   1:  PR[GP1:91,1] = PR[GP1:90,1] + 48.175;
   1:  PR[GP1:91,2] = PR[GP1:90,2] + 18.982;
   1:L PR[91] 10mm/sec CNT100;
   1:  PR[GP1:91,1] = PR[GP1:90,1] + 43.044;
   1:  PR[GP1:91,2] = PR[GP1:90,2] + 27.550;
   1:L PR[91] 10mm/sec CNT100;
   1:  PR[GP1:91,1] = PR[GP1:90,1] + 39.834;
   1:  PR[GP1:91,2] = PR[GP1:90,2] + 31.417;
   1:L PR[91] 10mm/sec CNT100;
   1:  PR[GP1:91,1] = PR[GP1:90,1] + 32.306;
   1:  PR[GP1:91,2] = PR[GP1:90,2] + 37.456;
   1:L PR[91] 10mm/sec CNT100;
   1:  PR[GP1:91,1] = PR[GP1:90,1] + 28.401;
   1:  PR[GP1:91,2] = PR[GP1:90,2] + 40.222;
   1:L PR[91] 10mm/sec CNT100;
   1:  PR[GP1:91,1] = PR[GP1:90,1] + 23.934;
   1:  PR[GP1:91,2] = PR[GP1:90,2] + 41.952;
   1:L PR[91] 10mm/sec CNT100;
   1:  PR[GP1:91,1] = PR[GP1:90,1] + 14.950;
   1:  PR[GP1:91,2] = PR[GP1:90,2] + 44.976;
   1:L PR[91] 10mm/sec CNT100;
   1:  PR[GP1:91,1] = PR[GP1:90,1] + 9.867;
   1:  PR[GP1:91,2] = PR[GP1:90,2] + 45.606;
   1:L PR[91] 10mm/sec CNT100;
   1:  PR[GP1:91,1] = PR[GP1:90,1] + 0.933;
   1:  PR[GP1:91,2] = PR[GP1:90,2] + 45.414;
   1:L PR[91] 10mm/sec CNT100;
   1:  PR[GP1:91,1] = PR[GP1:90,1] + -0.069;
   1:  PR[GP1:91,2] = PR[GP1:90,2] + 45.753;
   1:  PR[GP1:91,3] = PR[GP1:90,3] + 114.380;
   1:L PR[91] 10mm/sec CNT100;
   1:  PR[GP1:91,1] = PR[GP1:90,1] + -8.239;
   1:  PR[GP1:91,2] = PR[GP1:90,2] + 45.929;
   1:L PR[91] 10mm/sec CNT100;
   1:  PR[GP1:91,1] = PR[GP1:90,1] + -13.918;
   1:  PR[GP1:91,2] = PR[GP1:90,2] + 45.225;
   1:L PR[91] 10mm/sec CNT100;
   1:  PR[GP1:91,1] = PR[GP1:90,1] + -22.131;
   1:  PR[GP1:91,2] = PR[GP1:90,2] + 42.461;
   1:L PR[91] 10mm/sec CNT100;
   1:  PR[GP1:91,1] = PR[GP1:90,1] + -27.169;
   1:  PR[GP1:91,2] = PR[GP1:90,2] + 40.508;
   1:L PR[91] 10mm/sec CNT100;
   1:  PR[GP1:91,1] = PR[GP1:90,1] + -34.286;
   1:  PR[GP1:91,2] = PR[GP1:90,2] + 34.822;
   1:L PR[91] 10mm/sec CNT100;
   1:  PR[GP1:91,1] = PR[GP1:90,1] + -38.499;
   1:  PR[GP1:91,2] = PR[GP1:90,2] + 31.839;
   1:L PR[91] 10mm/sec CNT100;
   1:  PR[GP1:91,1] = PR[GP1:90,1] + -42.170;
   1:  PR[GP1:91,2] = PR[GP1:90,2] + 27.417;
   1:L PR[91] 10mm/sec CNT100;
   1:  PR[GP1:91,1] = PR[GP1:90,1] + -46.861;
   1:  PR[GP1:91,2] = PR[GP1:90,2] + 19.580;
   1:L PR[91] 10mm/sec CNT100;
   1:  PR[GP1:91,1] = PR[GP1:90,1] + -49.099;
   1:  PR[GP1:91,2] = PR[GP1:90,2] + 14.512;
   1:L PR[91] 10mm/sec CNT100;
   1:  PR[GP1:91,1] = PR[GP1:90,1] + -50.765;
   1:  PR[GP1:91,2] = PR[GP1:90,2] + 5.371;
   1:L PR[91] 10mm/sec CNT100;
   1:  PR[GP1:91,1] = PR[GP1:90,1] + -51.513;
   1:  PR[GP1:91,2] = PR[GP1:90,2] + 0.008;
   1:L PR[91] 10mm/sec CNT100;
   1:  PR[GP1:91,1] = PR[GP1:90,1] + -49.864;
   1:  PR[GP1:91,2] = PR[GP1:90,2] + -9.008;
   1:L PR[91] 10mm/sec CNT100;
   1:  PR[GP1:91,1] = PR[GP1:90,1] + -49.094;
   1:  PR[GP1:91,2] = PR[GP1:90,2] + -14.532;
   1:L PR[91] 10mm/sec CNT100;
   1:  PR[GP1:91,1] = PR[GP1:90,1] + -46.862;
   1:  PR[GP1:91,2] = PR[GP1:90,2] + -19.588;
   1:L PR[91] 10mm/sec CNT100;
   1:  PR[GP1:91,1] = PR[GP1:90,1] + -42.171;
   1:  PR[GP1:91,2] = PR[GP1:90,2] + -27.425;
   1:L PR[91] 10mm/sec CNT100;
   1:  PR[GP1:91,1] = PR[GP1:90,1] + -38.488;
   1:  PR[GP1:91,2] = PR[GP1:90,2] + -31.861;
   1:L PR[91] 10mm/sec CNT100;
   1:  PR[GP1:91,1] = PR[GP1:90,1] + -31.608;
   1:  PR[GP1:91,2] = PR[GP1:90,2] + -37.380;
   1:L PR[91] 10mm/sec CNT100;
   1:  PR[GP1:91,1] = PR[GP1:90,1] + -27.187;
   1:  PR[GP1:91,2] = PR[GP1:90,2] + -40.510;
   1:L PR[91] 10mm/sec CNT100;
   1:  PR[GP1:91,1] = PR[GP1:90,1] + -22.133;
   1:  PR[GP1:91,2] = PR[GP1:90,2] + -42.469;
   1:L PR[91] 10mm/sec CNT100;
   1:  PR[GP1:91,1] = PR[GP1:90,1] + -13.920;
   1:  PR[GP1:91,2] = PR[GP1:90,2] + -45.233;
   1:L PR[91] 10mm/sec CNT100;
   1:  PR[GP1:91,1] = PR[GP1:90,1] + -8.241;
   1:  PR[GP1:91,2] = PR[GP1:90,2] + -45.937;
   1:L PR[91] 10mm/sec CNT100;
   1:  PR[GP1:91,1] = PR[GP1:90,1] + -0.070;
   1:  PR[GP1:91,2] = PR[GP1:90,2] + -45.762;
   1:L PR[91] 10mm/sec CNT100;
   1:  PR[GP1:91,1] = PR[GP1:90,1] + 0.889;
   1:L PR[91] 10mm/sec CNT100;
   1:  PR[GP1:91,1] = PR[GP1:90,1] + 9.061;
   1:  PR[GP1:91,2] = PR[GP1:90,2] + -45.937;
   1:L PR[91] 10mm/sec CNT100;
   1:  PR[GP1:91,1] = PR[GP1:90,1] + 14.741;
   1:  PR[GP1:91,2] = PR[GP1:90,2] + -45.234;
   1:L PR[91] 10mm/sec CNT100;
   1:  PR[GP1:91,1] = PR[GP1:90,1] + 22.954;
   1:  PR[GP1:91,2] = PR[GP1:90,2] + -42.469;
   1:L PR[91] 10mm/sec CNT100;
   1:  PR[GP1:91,1] = PR[GP1:90,1] + 27.992;
   1:  PR[GP1:91,2] = PR[GP1:90,2] + -40.516;
   1:L PR[91] 10mm/sec CNT100;
   1:  PR[GP1:91,1] = PR[GP1:90,1] + 35.108;
   1:  PR[GP1:91,2] = PR[GP1:90,2] + -34.829;
   1:L PR[91] 10mm/sec CNT100;
   1:  PR[GP1:91,1] = PR[GP1:90,1] + 39.322;
   1:  PR[GP1:91,2] = PR[GP1:90,2] + -31.845;
   1:L PR[91] 10mm/sec CNT100;
   1:  PR[GP1:91,1] = PR[GP1:90,1] + 42.992;
   1:  PR[GP1:91,2] = PR[GP1:90,2] + -27.423;
   1:L PR[91] 10mm/sec CNT100;
   1:  PR[GP1:91,1] = PR[GP1:90,1] + 47.683;
   1:  PR[GP1:91,2] = PR[GP1:90,2] + -19.591;
   1:L PR[91] 10mm/sec CNT100;
   1:  PR[GP1:91,1] = PR[GP1:90,1] + 49.920;
   1:  PR[GP1:91,2] = PR[GP1:90,2] + -14.523;
   1:L PR[91] 10mm/sec CNT100;
   1:  PR[GP1:91,1] = PR[GP1:90,1] + 51.586;
   1:  PR[GP1:91,2] = PR[GP1:90,2] + -5.380;
   1:L PR[91] 10mm/sec CNT100;
   1:  PR[GP1:91,1] = PR[GP1:90,1] + 52.334;
   1:  PR[GP1:91,2] = PR[GP1:90,2] + -0.017;
   1:L PR[91] 10mm/sec CNT100;
   1:  PR[GP1:91,1] = PR[GP1:90,1] + 50.685;
   1:  PR[GP1:91,2] = PR[GP1:90,2] + 9.003;
   1:L PR[91] 10mm/sec CNT100;
   1:  PR[GP1:91,1] = PR[GP1:90,1] + 49.914;
   1:  PR[GP1:91,2] = PR[GP1:90,2] + 14.527;
   1:L PR[91] 10mm/sec CNT100;
   1:  PR[GP1:91,1] = PR[GP1:90,1] + 47.682;
   1:  PR[GP1:91,2] = PR[GP1:90,2] + 19.583;
   1:L PR[91] 10mm/sec CNT100;
   1:  PR[GP1:91,1] = PR[GP1:90,1] + 42.991;
   1:  PR[GP1:91,2] = PR[GP1:90,2] + 27.415;
   1:L PR[91] 10mm/sec CNT100;
   1:  PR[GP1:91,1] = PR[GP1:90,1] + 39.310;
   1:  PR[GP1:91,2] = PR[GP1:90,2] + 31.851;
   1:L PR[91] 10mm/sec CNT100;
   1:  PR[GP1:91,1] = PR[GP1:90,1] + 32.429;
   1:  PR[GP1:91,2] = PR[GP1:90,2] + 37.371;
   1:L PR[91] 10mm/sec CNT100;
   1:  PR[GP1:91,1] = PR[GP1:90,1] + 28.007;
   1:  PR[GP1:91,2] = PR[GP1:90,2] + 40.502;
   1:L PR[91] 10mm/sec CNT100;
   1:  PR[GP1:91,1] = PR[GP1:90,1] + 22.952;
   1:  PR[GP1:91,2] = PR[GP1:90,2] + 42.461;
   1:L PR[91] 10mm/sec CNT100;
   1:  PR[GP1:91,1] = PR[GP1:90,1] + 14.739;
   1:  PR[GP1:91,2] = PR[GP1:90,2] + 45.225;
   1:L PR[91] 10mm/sec CNT100;
   1:  PR[GP1:91,1] = PR[GP1:90,1] + 9.059;
   1:  PR[GP1:91,2] = PR[GP1:90,2] + 45.928;
   1:L PR[91] 10mm/sec CNT100;
   1:  PR[GP1:91,1] = PR[GP1:90,1] + 0.889;
   1:  PR[GP1:91,2] = PR[GP1:90,2] + 45.753;
   1:L PR[91] 10mm/sec CNT100;
   1:  PR[GP1:91,1] = PR[GP1:90,1] + -0.025;
   1:  PR[GP1:91,2] = PR[GP1:90,2] + 46.092;
   1:  PR[GP1:91,3] = PR[GP1:90,3] + 115.710;
   1:L PR[91] 10mm/sec CNT100;
   1:  PR[GP1:91,1] = PR[GP1:90,1] + -7.431;
   1:  PR[GP1:91,2] = PR[GP1:90,2] + 46.251;
   1:L PR[91] 10mm/sec CNT100;
   1:  PR[GP1:91,1] = PR[GP1:90,1] + -13.708;
   1:  PR[GP1:91,2] = PR[GP1:90,2] + 45.474;
   1:L PR[91] 10mm/sec CNT100;
   1:  PR[GP1:91,1] = PR[GP1:90,1] + -21.150;
   1:  PR[GP1:91,2] = PR[GP1:90,2] + 42.969;
   1:L PR[91] 10mm/sec CNT100;
   1:  PR[GP1:91,1] = PR[GP1:90,1] + -26.776;
   1:  PR[GP1:91,2] = PR[GP1:90,2] + 40.789;
   1:L PR[91] 10mm/sec CNT100;
   1:  PR[GP1:91,1] = PR[GP1:90,1] + -33.225;
   1:  PR[GP1:91,2] = PR[GP1:90,2] + 35.636;
   1:L PR[91] 10mm/sec CNT100;
   1:  PR[GP1:91,1] = PR[GP1:90,1] + -37.975;
   1:  PR[GP1:91,2] = PR[GP1:90,2] + 32.273;
   1:L PR[91] 10mm/sec CNT100;
   1:  PR[GP1:91,1] = PR[GP1:90,1] + -42.118;
   1:  PR[GP1:91,2] = PR[GP1:90,2] + 27.282;
   1:L PR[91] 10mm/sec CNT100;
   1:  PR[GP1:91,1] = PR[GP1:90,1] + -46.369;
   1:  PR[GP1:91,2] = PR[GP1:90,2] + 20.181;
   1:L PR[91] 10mm/sec CNT100;
   1:  PR[GP1:91,1] = PR[GP1:90,1] + -48.913;
   1:  PR[GP1:91,2] = PR[GP1:90,2] + 14.418;
   1:L PR[91] 10mm/sec CNT100;
   1:  PR[GP1:91,1] = PR[GP1:90,1] + -50.423;
   1:  PR[GP1:91,2] = PR[GP1:90,2] + 6.136;
   1:L PR[91] 10mm/sec CNT100;
   1:  PR[GP1:91,1] = PR[GP1:90,1] + -51.278;
   1:  PR[GP1:91,2] = PR[GP1:90,2] + 0.008;
   1:L PR[91] 10mm/sec CNT100;
   1:  PR[GP1:91,1] = PR[GP1:90,1] + -49.784;
   1:  PR[GP1:91,2] = PR[GP1:90,2] + -8.161;
   1:L PR[91] 10mm/sec CNT100;
   1:  PR[GP1:91,1] = PR[GP1:90,1] + -48.908;
   1:  PR[GP1:91,2] = PR[GP1:90,2] + -14.438;
   1:L PR[91] 10mm/sec CNT100;
   1:  PR[GP1:91,1] = PR[GP1:90,1] + -46.369;
   1:  PR[GP1:91,2] = PR[GP1:90,2] + -20.190;
   1:L PR[91] 10mm/sec CNT100;
   1:  PR[GP1:91,1] = PR[GP1:90,1] + -42.119;
   1:  PR[GP1:91,2] = PR[GP1:90,2] + -27.290;
   1:L PR[91] 10mm/sec CNT100;
   1:  PR[GP1:91,1] = PR[GP1:90,1] + -37.964;
   1:  PR[GP1:91,2] = PR[GP1:90,2] + -32.295;
   1:L PR[91] 10mm/sec CNT100;
   1:  PR[GP1:91,1] = PR[GP1:90,1] + -31.730;
   1:  PR[GP1:91,2] = PR[GP1:90,2] + -37.295;
   1:L PR[91] 10mm/sec CNT100;
   1:  PR[GP1:91,1] = PR[GP1:90,1] + -26.794;
   1:  PR[GP1:91,2] = PR[GP1:90,2] + -40.790;
   1:L PR[91] 10mm/sec CNT100;
   1:  PR[GP1:91,1] = PR[GP1:90,1] + -21.151;
   1:  PR[GP1:91,2] = PR[GP1:90,2] + -42.977;
   1:L PR[91] 10mm/sec CNT100;
   1:  PR[GP1:91,1] = PR[GP1:90,1] + -13.710;
   1:  PR[GP1:91,2] = PR[GP1:90,2] + -45.482;
   1:L PR[91] 10mm/sec CNT100;
   1:  PR[GP1:91,1] = PR[GP1:90,1] + -7.433;
   1:  PR[GP1:91,2] = PR[GP1:90,2] + -46.260;
   1:L PR[91] 10mm/sec CNT100;
   1:  PR[GP1:91,1] = PR[GP1:90,1] + -0.026;
   1:  PR[GP1:91,2] = PR[GP1:90,2] + -46.101;
   1:L PR[91] 10mm/sec CNT100;
   1:  PR[GP1:91,1] = PR[GP1:90,1] + 0.845;
   1:L PR[91] 10mm/sec CNT100;
   1:  PR[GP1:91,1] = PR[GP1:90,1] + 8.253;
   1:  PR[GP1:91,2] = PR[GP1:90,2] + -46.260;
   1:L PR[91] 10mm/sec CNT100;
   1:  PR[GP1:91,1] = PR[GP1:90,1] + 14.530;
   1:  PR[GP1:91,2] = PR[GP1:90,2] + -45.482;
   1:L PR[91] 10mm/sec CNT100;
   1:  PR[GP1:91,1] = PR[GP1:90,1] + 21.972;
   1:  PR[GP1:91,2] = PR[GP1:90,2] + -42.977;
   1:L PR[91] 10mm/sec CNT100;
   1:  PR[GP1:91,1] = PR[GP1:90,1] + 27.599;
   1:  PR[GP1:91,2] = PR[GP1:90,2] + -40.797;
   1:L PR[91] 10mm/sec CNT100;
   1:  PR[GP1:91,1] = PR[GP1:90,1] + 34.046;
   1:  PR[GP1:91,2] = PR[GP1:90,2] + -35.643;
   1:L PR[91] 10mm/sec CNT100;
   1:  PR[GP1:91,1] = PR[GP1:90,1] + 38.798;
   1:  PR[GP1:91,2] = PR[GP1:90,2] + -32.278;
   1:L PR[91] 10mm/sec CNT100;
   1:  PR[GP1:91,1] = PR[GP1:90,1] + 42.940;
   1:  PR[GP1:91,2] = PR[GP1:90,2] + -27.288;
   1:L PR[91] 10mm/sec CNT100;
   1:  PR[GP1:91,1] = PR[GP1:90,1] + 47.190;
   1:  PR[GP1:91,2] = PR[GP1:90,2] + -20.192;
   1:L PR[91] 10mm/sec CNT100;
   1:  PR[GP1:91,1] = PR[GP1:90,1] + 49.734;
   1:  PR[GP1:91,2] = PR[GP1:90,2] + -14.429;
   1:L PR[91] 10mm/sec CNT100;
   1:  PR[GP1:91,1] = PR[GP1:90,1] + 51.244;
   1:  PR[GP1:91,2] = PR[GP1:90,2] + -6.144;
   1:L PR[91] 10mm/sec CNT100;
   1:  PR[GP1:91,1] = PR[GP1:90,1] + 52.098;
   1:  PR[GP1:91,2] = PR[GP1:90,2] + -0.017;
   1:L PR[91] 10mm/sec CNT100;
   1:  PR[GP1:91,1] = PR[GP1:90,1] + 50.604;
   1:  PR[GP1:91,2] = PR[GP1:90,2] + 8.155;
   1:L PR[91] 10mm/sec CNT100;
   1:  PR[GP1:91,1] = PR[GP1:90,1] + 49.729;
   1:  PR[GP1:91,2] = PR[GP1:90,2] + 14.432;
   1:L PR[91] 10mm/sec CNT100;
   1:  PR[GP1:91,1] = PR[GP1:90,1] + 47.190;
   1:  PR[GP1:91,2] = PR[GP1:90,2] + 20.183;
   1:L PR[91] 10mm/sec CNT100;
   1:  PR[GP1:91,1] = PR[GP1:90,1] + 42.939;
   1:  PR[GP1:91,2] = PR[GP1:90,2] + 27.280;
   1:L PR[91] 10mm/sec CNT100;
   1:  PR[GP1:91,1] = PR[GP1:90,1] + 38.785;
   1:  PR[GP1:91,2] = PR[GP1:90,2] + 32.284;
   1:L PR[91] 10mm/sec CNT100;
   1:  PR[GP1:91,1] = PR[GP1:90,1] + 32.551;
   1:  PR[GP1:91,2] = PR[GP1:90,2] + 37.286;
   1:L PR[91] 10mm/sec CNT100;
   1:  PR[GP1:91,1] = PR[GP1:90,1] + 27.614;
   1:  PR[GP1:91,2] = PR[GP1:90,2] + 40.782;
   1:L PR[91] 10mm/sec CNT100;
   1:  PR[GP1:91,1] = PR[GP1:90,1] + 21.970;
   1:  PR[GP1:91,2] = PR[GP1:90,2] + 42.969;
   1:L PR[91] 10mm/sec CNT100;
   1:  PR[GP1:91,1] = PR[GP1:90,1] + 14.528;
   1:  PR[GP1:91,2] = PR[GP1:90,2] + 45.474;
   1:L PR[91] 10mm/sec CNT100;
   1:  PR[GP1:91,1] = PR[GP1:90,1] + 8.251;
   1:  PR[GP1:91,2] = PR[GP1:90,2] + 46.251;
   1:L PR[91] 10mm/sec CNT100;
   1:  PR[GP1:91,1] = PR[GP1:90,1] + 0.845;
   1:  PR[GP1:91,2] = PR[GP1:90,2] + 46.092;
   1:L PR[91] 10mm/sec CNT100;
   1:  PR[GP1:91,1] = PR[GP1:90,1] + 0.019;
   1:  PR[GP1:91,2] = PR[GP1:90,2] + 46.431;
   1:  PR[GP1:91,3] = PR[GP1:90,3] + 117.040;
   1:L PR[91] 10mm/sec CNT100;
   1:  PR[GP1:91,1] = PR[GP1:90,1] + -6.623;
   1:  PR[GP1:91,2] = PR[GP1:90,2] + 46.574;
   1:L PR[91] 10mm/sec CNT100;
   1:  PR[GP1:91,1] = PR[GP1:90,1] + -13.497;
   1:  PR[GP1:91,2] = PR[GP1:90,2] + 45.722;
   1:L PR[91] 10mm/sec CNT100;
   1:  PR[GP1:91,1] = PR[GP1:90,1] + -20.168;
   1:  PR[GP1:91,2] = PR[GP1:90,2] + 43.477;
   1:L PR[91] 10mm/sec CNT100;
   1:  PR[GP1:91,1] = PR[GP1:90,1] + -26.383;
   1:  PR[GP1:91,2] = PR[GP1:90,2] + 41.069;
   1:L PR[91] 10mm/sec CNT100;
   1:  PR[GP1:91,1] = PR[GP1:90,1] + -32.164;
   1:  PR[GP1:91,2] = PR[GP1:90,2] + 36.450;
   1:L PR[91] 10mm/sec CNT100;
   1:  PR[GP1:91,1] = PR[GP1:90,1] + -37.451;
   1:  PR[GP1:91,2] = PR[GP1:90,2] + 32.706;
   1:L PR[91] 10mm/sec CNT100;
   1:  PR[GP1:91,1] = PR[GP1:90,1] + -42.066;
   1:  PR[GP1:91,2] = PR[GP1:90,2] + 27.147;
   1:L PR[91] 10mm/sec CNT100;
   1:  PR[GP1:91,1] = PR[GP1:90,1] + -45.876;
   1:  PR[GP1:91,2] = PR[GP1:90,2] + 20.783;
   1:L PR[91] 10mm/sec CNT100;
   1:  PR[GP1:91,1] = PR[GP1:90,1] + -48.727;
   1:  PR[GP1:91,2] = PR[GP1:90,2] + 14.324;
   1:L PR[91] 10mm/sec CNT100;
   1:  PR[GP1:91,1] = PR[GP1:90,1] + -50.081;
   1:  PR[GP1:91,2] = PR[GP1:90,2] + 6.900;
   1:L PR[91] 10mm/sec CNT100;
   1:  PR[GP1:91,1] = PR[GP1:90,1] + -51.042;
   1:  PR[GP1:91,2] = PR[GP1:90,2] + 0.008;
   1:L PR[91] 10mm/sec CNT100;
   1:  PR[GP1:91,1] = PR[GP1:90,1] + -49.703;
   1:  PR[GP1:91,2] = PR[GP1:90,2] + -7.314;
   1:L PR[91] 10mm/sec CNT100;
   1:  PR[GP1:91,1] = PR[GP1:90,1] + -48.722;
   1:  PR[GP1:91,2] = PR[GP1:90,2] + -14.344;
   1:L PR[91] 10mm/sec CNT100;
   1:  PR[GP1:91,1] = PR[GP1:90,1] + -45.876;
   1:  PR[GP1:91,2] = PR[GP1:90,2] + -20.791;
   1:L PR[91] 10mm/sec CNT100;
   1:  PR[GP1:91,1] = PR[GP1:90,1] + -42.067;
   1:  PR[GP1:91,2] = PR[GP1:90,2] + -27.155;
   1:L PR[91] 10mm/sec CNT100;
   1:  PR[GP1:91,1] = PR[GP1:90,1] + -37.440;
   1:  PR[GP1:91,2] = PR[GP1:90,2] + -32.729;
   1:L PR[91] 10mm/sec CNT100;
   1:  PR[GP1:91,1] = PR[GP1:90,1] + -31.852;
   1:  PR[GP1:91,2] = PR[GP1:90,2] + -37.211;
   1:L PR[91] 10mm/sec CNT100;
   1:  PR[GP1:91,1] = PR[GP1:90,1] + -26.401;
   1:  PR[GP1:91,2] = PR[GP1:90,2] + -41.070;
   1:L PR[91] 10mm/sec CNT100;
   1:  PR[GP1:91,1] = PR[GP1:90,1] + -20.169;
   1:  PR[GP1:91,2] = PR[GP1:90,2] + -43.486;
   1:L PR[91] 10mm/sec CNT100;
   1:  PR[GP1:91,1] = PR[GP1:90,1] + -13.499;
   1:  PR[GP1:91,2] = PR[GP1:90,2] + -45.731;
   1:L PR[91] 10mm/sec CNT100;
   1:  PR[GP1:91,1] = PR[GP1:90,1] + -6.625;
   1:  PR[GP1:91,2] = PR[GP1:90,2] + -46.583;
   1:L PR[91] 10mm/sec CNT100;
   1:  PR[GP1:91,1] = PR[GP1:90,1] + 0.018;
   1:  PR[GP1:91,2] = PR[GP1:90,2] + -46.440;
   1:L PR[91] 10mm/sec CNT100;
   1:  PR[GP1:91,1] = PR[GP1:90,1] + 0.801;
   1:L PR[91] 10mm/sec CNT100;
   1:  PR[GP1:91,1] = PR[GP1:90,1] + 7.444;
   1:  PR[GP1:91,2] = PR[GP1:90,2] + -46.583;
   1:L PR[91] 10mm/sec CNT100;
   1:  PR[GP1:91,1] = PR[GP1:90,1] + 14.319;
   1:  PR[GP1:91,2] = PR[GP1:90,2] + -45.731;
   1:L PR[91] 10mm/sec CNT100;
   1:  PR[GP1:91,1] = PR[GP1:90,1] + 20.989;
   1:  PR[GP1:91,2] = PR[GP1:90,2] + -43.486;
   1:L PR[91] 10mm/sec CNT100;
   1:  PR[GP1:91,1] = PR[GP1:90,1] + 27.206;
   1:  PR[GP1:91,2] = PR[GP1:90,2] + -41.077;
   1:L PR[91] 10mm/sec CNT100;
   1:  PR[GP1:91,1] = PR[GP1:90,1] + 32.985;
   1:  PR[GP1:91,2] = PR[GP1:90,2] + -36.457;
   1:L PR[91] 10mm/sec CNT100;
   1:  PR[GP1:91,1] = PR[GP1:90,1] + 38.273;
   1:  PR[GP1:91,2] = PR[GP1:90,2] + -32.712;
   1:L PR[91] 10mm/sec CNT100;
   1:  PR[GP1:91,1] = PR[GP1:90,1] + 42.888;
   1:  PR[GP1:91,2] = PR[GP1:90,2] + -27.153;
   1:L PR[91] 10mm/sec CNT100;
   1:  PR[GP1:91,1] = PR[GP1:90,1] + 46.697;
   1:  PR[GP1:91,2] = PR[GP1:90,2] + -20.793;
   1:L PR[91] 10mm/sec CNT100;
   1:  PR[GP1:91,1] = PR[GP1:90,1] + 49.548;
   1:  PR[GP1:91,2] = PR[GP1:90,2] + -14.334;
   1:L PR[91] 10mm/sec CNT100;
   1:  PR[GP1:91,1] = PR[GP1:90,1] + 50.902;
   1:  PR[GP1:91,2] = PR[GP1:90,2] + -6.909;
   1:L PR[91] 10mm/sec CNT100;
   1:  PR[GP1:91,1] = PR[GP1:90,1] + 51.863;
   1:  PR[GP1:91,2] = PR[GP1:90,2] + -0.017;
   1:L PR[91] 10mm/sec CNT100;
   1:  PR[GP1:91,1] = PR[GP1:90,1] + 50.523;
   1:  PR[GP1:91,2] = PR[GP1:90,2] + 7.308;
   1:L PR[91] 10mm/sec CNT100;
   1:  PR[GP1:91,1] = PR[GP1:90,1] + 49.543;
   1:  PR[GP1:91,2] = PR[GP1:90,2] + 14.337;
   1:L PR[91] 10mm/sec CNT100;
   1:  PR[GP1:91,1] = PR[GP1:90,1] + 46.697;
   1:  PR[GP1:91,2] = PR[GP1:90,2] + 20.784;
   1:L PR[91] 10mm/sec CNT100;
   1:  PR[GP1:91,1] = PR[GP1:90,1] + 42.887;
   1:  PR[GP1:91,2] = PR[GP1:90,2] + 27.145;
   1:L PR[91] 10mm/sec CNT100;
   1:  PR[GP1:91,1] = PR[GP1:90,1] + 38.261;
   1:  PR[GP1:91,2] = PR[GP1:90,2] + 32.718;
   1:L PR[91] 10mm/sec CNT100;
   1:  PR[GP1:91,1] = PR[GP1:90,1] + 32.673;
   1:  PR[GP1:91,2] = PR[GP1:90,2] + 37.202;
   1:L PR[91] 10mm/sec CNT100;
   1:  PR[GP1:91,1] = PR[GP1:90,1] + 27.221;
   1:  PR[GP1:91,2] = PR[GP1:90,2] + 41.062;
   1:L PR[91] 10mm/sec CNT100;
   1:  PR[GP1:91,1] = PR[GP1:90,1] + 20.988;
   1:  PR[GP1:91,2] = PR[GP1:90,2] + 43.477;
   1:L PR[91] 10mm/sec CNT100;
   1:  PR[GP1:91,1] = PR[GP1:90,1] + 14.318;
   1:  PR[GP1:91,2] = PR[GP1:90,2] + 45.723;
   1:L PR[91] 10mm/sec CNT100;
   1:  PR[GP1:91,1] = PR[GP1:90,1] + 7.443;
   1:  PR[GP1:91,2] = PR[GP1:90,2] + 46.574;
   1:L PR[91] 10mm/sec CNT100;
   1:  PR[GP1:91,1] = PR[GP1:90,1] + 0.801;
   1:  PR[GP1:91,2] = PR[GP1:90,2] + 46.431;
   1:L PR[91] 10mm/sec CNT100;
   1:  PR[GP1:91,1] = PR[GP1:90,1] + 0.062;
   1:  PR[GP1:91,2] = PR[GP1:90,2] + 46.770;
   1:  PR[GP1:91,3] = PR[GP1:90,3] + 118.370;
   1:L PR[91] 10mm/sec CNT100;
   1:  PR[GP1:91,1] = PR[GP1:90,1] + -5.815;
   1:  PR[GP1:91,2] = PR[GP1:90,2] + 46.897;
   1:L PR[91] 10mm/sec CNT100;
   1:  PR[GP1:91,1] = PR[GP1:90,1] + -13.287;
   1:  PR[GP1:91,2] = PR[GP1:90,2] + 45.971;
   1:L PR[91] 10mm/sec CNT100;
   1:  PR[GP1:91,1] = PR[GP1:90,1] + -19.186;
   1:  PR[GP1:91,2] = PR[GP1:90,2] + 43.986;
   1:L PR[91] 10mm/sec CNT100;
   1:  PR[GP1:91,1] = PR[GP1:90,1] + -25.990;
   1:  PR[GP1:91,2] = PR[GP1:90,2] + 41.349;
   1:L PR[91] 10mm/sec CNT100;
   1:  PR[GP1:91,1] = PR[GP1:90,1] + -31.103;
   1:  PR[GP1:91,2] = PR[GP1:90,2] + 37.264;
   1:L PR[91] 10mm/sec CNT100;
   1:  PR[GP1:91,1] = PR[GP1:90,1] + -36.927;
   1:  PR[GP1:91,2] = PR[GP1:90,2] + 33.140;
   1:L PR[91] 10mm/sec CNT100;
   1:  PR[GP1:91,1] = PR[GP1:90,1] + -42.014;
   1:  PR[GP1:91,2] = PR[GP1:90,2] + 27.012;
   1:L PR[91] 10mm/sec CNT100;
   1:  PR[GP1:91,1] = PR[GP1:90,1] + -45.383;
   1:  PR[GP1:91,2] = PR[GP1:90,2] + 21.384;
   1:L PR[91] 10mm/sec CNT100;
   1:  PR[GP1:91,1] = PR[GP1:90,1] + -48.542;
   1:  PR[GP1:91,2] = PR[GP1:90,2] + 14.229;
   1:L PR[91] 10mm/sec CNT100;
   1:  PR[GP1:91,1] = PR[GP1:90,1] + -49.739;
   1:  PR[GP1:91,2] = PR[GP1:90,2] + 7.665;
   1:L PR[91] 10mm/sec CNT100;
   1:  PR[GP1:91,1] = PR[GP1:90,1] + -50.806;
   1:  PR[GP1:91,2] = PR[GP1:90,2] + 0.008;
   1:L PR[91] 10mm/sec CNT100;
   1:  PR[GP1:91,1] = PR[GP1:90,1] + -49.622;
   1:  PR[GP1:91,2] = PR[GP1:90,2] + -6.467;
   1:L PR[91] 10mm/sec CNT100;
   1:  PR[GP1:91,1] = PR[GP1:90,1] + -48.537;
   1:  PR[GP1:91,2] = PR[GP1:90,2] + -14.249;
   1:L PR[91] 10mm/sec CNT100;
   1:  PR[GP1:91,1] = PR[GP1:90,1] + -45.383;
   1:  PR[GP1:91,2] = PR[GP1:90,2] + -21.392;
   1:L PR[91] 10mm/sec CNT100;
   1:  PR[GP1:91,1] = PR[GP1:90,1] + -42.015;
   1:  PR[GP1:91,2] = PR[GP1:90,2] + -27.020;
   1:L PR[91] 10mm/sec CNT100;
   1:  PR[GP1:91,1] = PR[GP1:90,1] + -36.915;
   1:  PR[GP1:91,2] = PR[GP1:90,2] + -33.162;
   1:L PR[91] 10mm/sec CNT100;
   1:  PR[GP1:91,1] = PR[GP1:90,1] + -31.974;
   1:  PR[GP1:91,2] = PR[GP1:90,2] + -37.126;
   1:L PR[91] 10mm/sec CNT100;
   1:  PR[GP1:91,1] = PR[GP1:90,1] + -26.008;
   1:  PR[GP1:91,2] = PR[GP1:90,2] + -41.351;
   1:L PR[91] 10mm/sec CNT100;
   1:  PR[GP1:91,1] = PR[GP1:90,1] + -19.187;
   1:  PR[GP1:91,2] = PR[GP1:90,2] + -43.994;
   1:L PR[91] 10mm/sec CNT100;
   1:  PR[GP1:91,1] = PR[GP1:90,1] + -13.288;
   1:  PR[GP1:91,2] = PR[GP1:90,2] + -45.980;
   1:L PR[91] 10mm/sec CNT100;
   1:  PR[GP1:91,1] = PR[GP1:90,1] + -5.817;
   1:  PR[GP1:91,2] = PR[GP1:90,2] + -46.905;
   1:L PR[91] 10mm/sec CNT100;
   1:  PR[GP1:91,1] = PR[GP1:90,1] + 0.062;
   1:  PR[GP1:91,2] = PR[GP1:90,2] + -46.779;
   1:L PR[91] 10mm/sec CNT100;
   1:  PR[GP1:91,1] = PR[GP1:90,1] + 0.757;
   1:L PR[91] 10mm/sec CNT100;
   1:  PR[GP1:91,1] = PR[GP1:90,1] + 6.636;
   1:  PR[GP1:91,2] = PR[GP1:90,2] + -46.905;
   1:L PR[91] 10mm/sec CNT100;
   1:  PR[GP1:91,1] = PR[GP1:90,1] + 14.108;
   1:  PR[GP1:91,2] = PR[GP1:90,2] + -45.980;
   1:L PR[91] 10mm/sec CNT100;
   1:  PR[GP1:91,1] = PR[GP1:90,1] + 20.007;
   1:  PR[GP1:91,2] = PR[GP1:90,2] + -43.994;
   1:L PR[91] 10mm/sec CNT100;
   1:  PR[GP1:91,1] = PR[GP1:90,1] + 26.812;
   1:  PR[GP1:91,2] = PR[GP1:90,2] + -41.357;
   1:L PR[91] 10mm/sec CNT100;
   1:  PR[GP1:91,1] = PR[GP1:90,1] + 31.924;
   1:  PR[GP1:91,2] = PR[GP1:90,2] + -37.271;
   1:L PR[91] 10mm/sec CNT100;
   1:  PR[GP1:91,1] = PR[GP1:90,1] + 37.749;
   1:  PR[GP1:91,2] = PR[GP1:90,2] + -33.146;
   1:L PR[91] 10mm/sec CNT100;
   1:  PR[GP1:91,1] = PR[GP1:90,1] + 42.836;
   1:  PR[GP1:91,2] = PR[GP1:90,2] + -27.018;
   1:L PR[91] 10mm/sec CNT100;
   1:  PR[GP1:91,1] = PR[GP1:90,1] + 46.204;
   1:  PR[GP1:91,2] = PR[GP1:90,2] + -21.394;
   1:L PR[91] 10mm/sec CNT100;
   1:  PR[GP1:91,1] = PR[GP1:90,1] + 49.363;
   1:  PR[GP1:91,2] = PR[GP1:90,2] + -14.240;
   1:L PR[91] 10mm/sec CNT100;
   1:  PR[GP1:91,1] = PR[GP1:90,1] + 50.559;
   1:  PR[GP1:91,2] = PR[GP1:90,2] + -7.673;
   1:L PR[91] 10mm/sec CNT100;
   1:  PR[GP1:91,1] = PR[GP1:90,1] + 51.627;
   1:  PR[GP1:91,2] = PR[GP1:90,2] + -0.017;
   1:L PR[91] 10mm/sec CNT100;
   1:  PR[GP1:91,1] = PR[GP1:90,1] + 50.443;
   1:  PR[GP1:91,2] = PR[GP1:90,2] + 6.460;
   1:L PR[91] 10mm/sec CNT100;
   1:  PR[GP1:91,1] = PR[GP1:90,1] + 49.357;
   1:  PR[GP1:91,2] = PR[GP1:90,2] + 14.243;
   1:L PR[91] 10mm/sec CNT100;
   1:  PR[GP1:91,1] = PR[GP1:90,1] + 46.204;
   1:  PR[GP1:91,2] = PR[GP1:90,2] + 21.385;
   1:L PR[91] 10mm/sec CNT100;
   1:  PR[GP1:91,1] = PR[GP1:90,1] + 42.835;
   1:  PR[GP1:91,2] = PR[GP1:90,2] + 27.010;
   1:L PR[91] 10mm/sec CNT100;
   1:  PR[GP1:91,1] = PR[GP1:90,1] + 37.737;
   1:  PR[GP1:91,2] = PR[GP1:90,2] + 33.152;
   1:L PR[91] 10mm/sec CNT100;
   1:  PR[GP1:91,1] = PR[GP1:90,1] + 32.795;
   1:  PR[GP1:91,2] = PR[GP1:90,2] + 37.117;
   1:L PR[91] 10mm/sec CNT100;
   1:  PR[GP1:91,1] = PR[GP1:90,1] + 26.828;
   1:  PR[GP1:91,2] = PR[GP1:90,2] + 41.342;
   1:L PR[91] 10mm/sec CNT100;
   1:  PR[GP1:91,1] = PR[GP1:90,1] + 20.006;
   1:  PR[GP1:91,2] = PR[GP1:90,2] + 43.986;
   1:L PR[91] 10mm/sec CNT100;
   1:  PR[GP1:91,1] = PR[GP1:90,1] + 14.107;
   1:  PR[GP1:91,2] = PR[GP1:90,2] + 45.971;
   1:L PR[91] 10mm/sec CNT100;
   1:  PR[GP1:91,1] = PR[GP1:90,1] + 6.634;
   1:  PR[GP1:91,2] = PR[GP1:90,2] + 46.897;
   1:L PR[91] 10mm/sec CNT100;
   1:  PR[GP1:91,1] = PR[GP1:90,1] + 0.756;
   1:  PR[GP1:91,2] = PR[GP1:90,2] + 46.770;
   1:L PR[91] 10mm/sec CNT100;
   1:  PR[GP1:91,1] = PR[GP1:90,1] + 0.106;
   1:  PR[GP1:91,2] = PR[GP1:90,2] + 47.109;
   1:  PR[GP1:91,3] = PR[GP1:90,3] + 119.700;
   1:L PR[91] 10mm/sec CNT100;
   1:  PR[GP1:91,1] = PR[GP1:90,1] + -5.007;
   1:  PR[GP1:91,2] = PR[GP1:90,2] + 47.219;
   1:L PR[91] 10mm/sec CNT100;
   1:  PR[GP1:91,1] = PR[GP1:90,1] + -13.076;
   1:  PR[GP1:91,2] = PR[GP1:90,2] + 46.220;
   1:L PR[91] 10mm/sec CNT100;
   1:  PR[GP1:91,1] = PR[GP1:90,1] + -18.204;
   1:  PR[GP1:91,2] = PR[GP1:90,2] + 44.494;
   1:L PR[91] 10mm/sec CNT100;
   1:  PR[GP1:91,1] = PR[GP1:90,1] + -25.597;
   1:  PR[GP1:91,2] = PR[GP1:90,2] + 41.629;
   1:L PR[91] 10mm/sec CNT100;
   1:  PR[GP1:91,1] = PR[GP1:90,1] + -30.041;
   1:  PR[GP1:91,2] = PR[GP1:90,2] + 38.078;
   1:L PR[91] 10mm/sec CNT100;
   1:  PR[GP1:91,1] = PR[GP1:90,1] + -36.402;
   1:  PR[GP1:91,2] = PR[GP1:90,2] + 33.574;
   1:L PR[91] 10mm/sec CNT100;
   1:  PR[GP1:91,1] = PR[GP1:90,1] + -41.962;
   1:  PR[GP1:91,2] = PR[GP1:90,2] + 26.877;
   1:L PR[91] 10mm/sec CNT100;
   1:  PR[GP1:91,1] = PR[GP1:90,1] + -44.890;
   1:  PR[GP1:91,2] = PR[GP1:90,2] + 21.985;
   1:L PR[91] 10mm/sec CNT100;
   1:  PR[GP1:91,1] = PR[GP1:90,1] + -48.356;
   1:  PR[GP1:91,2] = PR[GP1:90,2] + 14.135;
   1:L PR[91] 10mm/sec CNT100;
   1:  PR[GP1:91,1] = PR[GP1:90,1] + -49.396;
   1:  PR[GP1:91,2] = PR[GP1:90,2] + 8.429;
   1:L PR[91] 10mm/sec CNT100;
   1:  PR[GP1:91,1] = PR[GP1:90,1] + -50.571;
   1:  PR[GP1:91,2] = PR[GP1:90,2] + 0.008;
   1:L PR[91] 10mm/sec CNT100;
   1:  PR[GP1:91,1] = PR[GP1:90,1] + -49.541;
   1:  PR[GP1:91,2] = PR[GP1:90,2] + -5.619;
   1:L PR[91] 10mm/sec CNT100;
   1:  PR[GP1:91,1] = PR[GP1:90,1] + -48.351;
   1:  PR[GP1:91,2] = PR[GP1:90,2] + -14.155;
   1:L PR[91] 10mm/sec CNT100;
   1:  PR[GP1:91,1] = PR[GP1:90,1] + -44.891;
   1:  PR[GP1:91,2] = PR[GP1:90,2] + -21.993;
   1:L PR[91] 10mm/sec CNT100;
   1:  PR[GP1:91,1] = PR[GP1:90,1] + -41.963;
   1:  PR[GP1:91,2] = PR[GP1:90,2] + -26.885;
   1:L PR[91] 10mm/sec CNT100;
   1:  PR[GP1:91,1] = PR[GP1:90,1] + -36.391;
   1:  PR[GP1:91,2] = PR[GP1:90,2] + -33.596;
   1:L PR[91] 10mm/sec CNT100;
   1:  PR[GP1:91,1] = PR[GP1:90,1] + -32.096;
   1:  PR[GP1:91,2] = PR[GP1:90,2] + -37.041;
   1:L PR[91] 10mm/sec CNT100;
   1:  PR[GP1:91,1] = PR[GP1:90,1] + -25.615;
   1:  PR[GP1:91,2] = PR[GP1:90,2] + -41.631;
   1:L PR[91] 10mm/sec CNT100;
   1:  PR[GP1:91,1] = PR[GP1:90,1] + -18.205;
   1:  PR[GP1:91,2] = PR[GP1:90,2] + -44.502;
   1:L PR[91] 10mm/sec CNT100;
   1:  PR[GP1:91,1] = PR[GP1:90,1] + -13.077;
   1:  PR[GP1:91,2] = PR[GP1:90,2] + -46.228;
   1:L PR[91] 10mm/sec CNT100;
   1:  PR[GP1:91,1] = PR[GP1:90,1] + -5.008;
   1:  PR[GP1:91,2] = PR[GP1:90,2] + -47.228;
   1:L PR[91] 10mm/sec CNT100;
   1:  PR[GP1:91,1] = PR[GP1:90,1] + 0.106;
   1:  PR[GP1:91,2] = PR[GP1:90,2] + -47.118;
   1:L PR[91] 10mm/sec CNT100;
   1:  PR[GP1:91,1] = PR[GP1:90,1] + 0.713;
   1:L PR[91] 10mm/sec CNT100;
   1:  PR[GP1:91,1] = PR[GP1:90,1] + 5.827;
   1:  PR[GP1:91,2] = PR[GP1:90,2] + -47.228;
   1:L PR[91] 10mm/sec CNT100;
   1:  PR[GP1:91,1] = PR[GP1:90,1] + 13.897;
   1:  PR[GP1:91,2] = PR[GP1:90,2] + -46.229;
   1:L PR[91] 10mm/sec CNT100;
   1:  PR[GP1:91,1] = PR[GP1:90,1] + 19.025;
   1:  PR[GP1:91,2] = PR[GP1:90,2] + -44.502;
   1:L PR[91] 10mm/sec CNT100;
   1:  PR[GP1:91,1] = PR[GP1:90,1] + 26.419;
   1:  PR[GP1:91,2] = PR[GP1:90,2] + -41.637;
   1:L PR[91] 10mm/sec CNT100;
   1:  PR[GP1:91,1] = PR[GP1:90,1] + 30.863;
   1:  PR[GP1:91,2] = PR[GP1:90,2] + -38.085;
   1:L PR[91] 10mm/sec CNT100;
   1:  PR[GP1:91,1] = PR[GP1:90,1] + 37.225;
   1:  PR[GP1:91,2] = PR[GP1:90,2] + -33.580;
   1:L PR[91] 10mm/sec CNT100;
   1:  PR[GP1:91,1] = PR[GP1:90,1] + 42.784;
   1:  PR[GP1:91,2] = PR[GP1:90,2] + -26.883;
   1:L PR[91] 10mm/sec CNT100;
   1:  PR[GP1:91,1] = PR[GP1:90,1] + 45.712;
   1:  PR[GP1:91,2] = PR[GP1:90,2] + -21.994;
   1:L PR[91] 10mm/sec CNT100;
   1:  PR[GP1:91,1] = PR[GP1:90,1] + 49.177;
   1:  PR[GP1:91,2] = PR[GP1:90,2] + -14.145;
   1:L PR[91] 10mm/sec CNT100;
   1:  PR[GP1:91,1] = PR[GP1:90,1] + 50.217;
   1:  PR[GP1:91,2] = PR[GP1:90,2] + -8.438;
   1:L PR[91] 10mm/sec CNT100;
   1:  PR[GP1:91,1] = PR[GP1:90,1] + 51.391;
   1:  PR[GP1:91,2] = PR[GP1:90,2] + -0.017;
   1:L PR[91] 10mm/sec CNT100;
   1:  PR[GP1:91,1] = PR[GP1:90,1] + 50.362;
   1:  PR[GP1:91,2] = PR[GP1:90,2] + 5.613;
   1:L PR[91] 10mm/sec CNT100;
   1:  PR[GP1:91,1] = PR[GP1:90,1] + 49.172;
   1:  PR[GP1:91,2] = PR[GP1:90,2] + 14.148;
   1:L PR[91] 10mm/sec CNT100;
   1:  PR[GP1:91,1] = PR[GP1:90,1] + 45.712;
   1:  PR[GP1:91,2] = PR[GP1:90,2] + 21.986;
   1:L PR[91] 10mm/sec CNT100;
   1:  PR[GP1:91,1] = PR[GP1:90,1] + 42.783;
   1:  PR[GP1:91,2] = PR[GP1:90,2] + 26.875;
   1:L PR[91] 10mm/sec CNT100;
   1:  PR[GP1:91,1] = PR[GP1:90,1] + 37.213;
   1:  PR[GP1:91,2] = PR[GP1:90,2] + 33.586;
   1:L PR[91] 10mm/sec CNT100;
   1:  PR[GP1:91,1] = PR[GP1:90,1] + 32.917;
   1:  PR[GP1:91,2] = PR[GP1:90,2] + 37.032;
   1:L PR[91] 10mm/sec CNT100;
   1:  PR[GP1:91,1] = PR[GP1:90,1] + 26.435;
   1:  PR[GP1:91,2] = PR[GP1:90,2] + 41.622;
   1:L PR[91] 10mm/sec CNT100;
   1:  PR[GP1:91,1] = PR[GP1:90,1] + 19.024;
   1:  PR[GP1:91,2] = PR[GP1:90,2] + 44.494;
   1:L PR[91] 10mm/sec CNT100;
   1:  PR[GP1:91,1] = PR[GP1:90,1] + 13.896;
   1:  PR[GP1:91,2] = PR[GP1:90,2] + 46.220;
   1:L PR[91] 10mm/sec CNT100;
   1:  PR[GP1:91,1] = PR[GP1:90,1] + 5.826;
   1:  PR[GP1:91,2] = PR[GP1:90,2] + 47.219;
   1:L PR[91] 10mm/sec CNT100;
   1:  PR[GP1:91,1] = PR[GP1:90,1] + 0.712;
   1:  PR[GP1:91,2] = PR[GP1:90,2] + 47.109;
   1:L PR[91] 10mm/sec CNT100;
   1:  PR[GP1:91,1] = PR[GP1:90,1] + -4.199;
   1:  PR[GP1:91,2] = PR[GP1:90,2] + 47.542;
   1:  PR[GP1:91,3] = PR[GP1:90,3] + 121.030;
   1:L PR[91] 10mm/sec CNT100;
   1:  PR[GP1:91,1] = PR[GP1:90,1] + -12.865;
   1:  PR[GP1:91,2] = PR[GP1:90,2] + 46.468;
   1:L PR[91] 10mm/sec CNT100;
   1:  PR[GP1:91,1] = PR[GP1:90,1] + -17.222;
   1:  PR[GP1:91,2] = PR[GP1:90,2] + 45.002;
   1:L PR[91] 10mm/sec CNT100;
   1:  PR[GP1:91,1] = PR[GP1:90,1] + -25.204;
   1:  PR[GP1:91,2] = PR[GP1:90,2] + 41.909;
   1:L PR[91] 10mm/sec CNT100;
   1:  PR[GP1:91,1] = PR[GP1:90,1] + -28.980;
   1:  PR[GP1:91,2] = PR[GP1:90,2] + 38.892;
   1:L PR[91] 10mm/sec CNT100;
   1:  PR[GP1:91,1] = PR[GP1:90,1] + -35.878;
   1:  PR[GP1:91,2] = PR[GP1:90,2] + 34.007;
   1:L PR[91] 10mm/sec CNT100;
   1:  PR[GP1:91,1] = PR[GP1:90,1] + -41.910;
   1:  PR[GP1:91,2] = PR[GP1:90,2] + 26.742;
   1:L PR[91] 10mm/sec CNT100;
   1:  PR[GP1:91,1] = PR[GP1:90,1] + -44.398;
   1:  PR[GP1:91,2] = PR[GP1:90,2] + 22.586;
   1:L PR[91] 10mm/sec CNT100;
   1:  PR[GP1:91,1] = PR[GP1:90,1] + -48.170;
   1:  PR[GP1:91,2] = PR[GP1:90,2] + 14.041;
   1:L PR[91] 10mm/sec CNT100;
   1:  PR[GP1:91,1] = PR[GP1:90,1] + -49.054;
   1:  PR[GP1:91,2] = PR[GP1:90,2] + 9.194;
   1:L PR[91] 10mm/sec CNT100;
   1:  PR[GP1:91,1] = PR[GP1:90,1] + -50.335;
   1:  PR[GP1:91,2] = PR[GP1:90,2] + 0.008;
   1:L PR[91] 10mm/sec CNT100;
   1:  PR[GP1:91,1] = PR[GP1:90,1] + -49.461;
   1:  PR[GP1:91,2] = PR[GP1:90,2] + -4.772;
   1:L PR[91] 10mm/sec CNT100;
   1:  PR[GP1:91,1] = PR[GP1:90,1] + -48.165;
   1:  PR[GP1:91,2] = PR[GP1:90,2] + -14.061;
   1:L PR[91] 10mm/sec CNT100;
   1:  PR[GP1:91,1] = PR[GP1:90,1] + -44.398;
   1:  PR[GP1:91,2] = PR[GP1:90,2] + -22.595;
   1:L PR[91] 10mm/sec CNT100;
   1:  PR[GP1:91,1] = PR[GP1:90,1] + -41.911;
   1:  PR[GP1:91,2] = PR[GP1:90,2] + -26.750;
   1:L PR[91] 10mm/sec CNT100;
   1:  PR[GP1:91,1] = PR[GP1:90,1] + -35.867;
   1:  PR[GP1:91,2] = PR[GP1:90,2] + -34.030;
   1:L PR[91] 10mm/sec CNT100;
   1:  PR[GP1:91,1] = PR[GP1:90,1] + -32.218;
   1:  PR[GP1:91,2] = PR[GP1:90,2] + -36.956;
   1:L PR[91] 10mm/sec CNT100;
   1:  PR[GP1:91,1] = PR[GP1:90,1] + -25.221;
   1:  PR[GP1:91,2] = PR[GP1:90,2] + -41.911;
   1:L PR[91] 10mm/sec CNT100;
   1:  PR[GP1:91,1] = PR[GP1:90,1] + -17.223;
   1:  PR[GP1:91,2] = PR[GP1:90,2] + -45.011;
   1:L PR[91] 10mm/sec CNT100;
   1:  PR[GP1:91,1] = PR[GP1:90,1] + -12.867;
   1:  PR[GP1:91,2] = PR[GP1:90,2] + -46.477;
   1:L PR[91] 10mm/sec CNT100;
   1:  PR[GP1:91,1] = PR[GP1:90,1] + -4.200;
   1:  PR[GP1:91,2] = PR[GP1:90,2] + -47.551;
   1:L PR[91] 10mm/sec CNT100;
   1:  PR[GP1:91,1] = PR[GP1:90,1] + 0.156;
   1:  PR[GP1:91,2] = PR[GP1:90,2] + -47.457;
   1:L PR[91] 10mm/sec CNT100;
   1:  PR[GP1:91,1] = PR[GP1:90,1] + 5.018;
   1:  PR[GP1:91,2] = PR[GP1:90,2] + -47.551;
   1:L PR[91] 10mm/sec CNT100;
   1:  PR[GP1:91,1] = PR[GP1:90,1] + 13.686;
   1:  PR[GP1:91,2] = PR[GP1:90,2] + -46.477;
   1:L PR[91] 10mm/sec CNT100;
   1:  PR[GP1:91,1] = PR[GP1:90,1] + 18.043;
   1:  PR[GP1:91,2] = PR[GP1:90,2] + -45.011;
   1:L PR[91] 10mm/sec CNT100;
   1:  PR[GP1:91,1] = PR[GP1:90,1] + 26.026;
   1:  PR[GP1:91,2] = PR[GP1:90,2] + -41.917;
   1:L PR[91] 10mm/sec CNT100;
   1:  PR[GP1:91,1] = PR[GP1:90,1] + 29.801;
   1:  PR[GP1:91,2] = PR[GP1:90,2] + -38.899;
   1:L PR[91] 10mm/sec CNT100;
   1:  PR[GP1:91,1] = PR[GP1:90,1] + 36.701;
   1:  PR[GP1:91,2] = PR[GP1:90,2] + -34.014;
   1:L PR[91] 10mm/sec CNT100;
   1:  PR[GP1:91,1] = PR[GP1:90,1] + 42.732;
   1:  PR[GP1:91,2] = PR[GP1:90,2] + -26.749;
   1:L PR[91] 10mm/sec CNT100;
   1:  PR[GP1:91,1] = PR[GP1:90,1] + 45.219;
   1:  PR[GP1:91,2] = PR[GP1:90,2] + -22.595;
   1:L PR[91] 10mm/sec CNT100;
   1:  PR[GP1:91,1] = PR[GP1:90,1] + 48.991;
   1:  PR[GP1:91,2] = PR[GP1:90,2] + -14.051;
   1:L PR[91] 10mm/sec CNT100;
   1:  PR[GP1:91,1] = PR[GP1:90,1] + 49.875;
   1:  PR[GP1:91,2] = PR[GP1:90,2] + -9.202;
   1:L PR[91] 10mm/sec CNT100;
   1:  PR[GP1:91,1] = PR[GP1:90,1] + 51.156;
   1:  PR[GP1:91,2] = PR[GP1:90,2] + -0.017;
   1:L PR[91] 10mm/sec CNT100;
   1:  PR[GP1:91,1] = PR[GP1:90,1] + 50.281;
   1:  PR[GP1:91,2] = PR[GP1:90,2] + 4.765;
   1:L PR[91] 10mm/sec CNT100;
   1:  PR[GP1:91,1] = PR[GP1:90,1] + 48.986;
   1:  PR[GP1:91,2] = PR[GP1:90,2] + 14.054;
   1:L PR[91] 10mm/sec CNT100;
   1:  PR[GP1:91,1] = PR[GP1:90,1] + 45.219;
   1:  PR[GP1:91,2] = PR[GP1:90,2] + 22.587;
   1:L PR[91] 10mm/sec CNT100;
   1:  PR[GP1:91,1] = PR[GP1:90,1] + 42.731;
   1:  PR[GP1:91,2] = PR[GP1:90,2] + 26.740;
   1:L PR[91] 10mm/sec CNT100;
   1:  PR[GP1:91,1] = PR[GP1:90,1] + 36.689;
   1:  PR[GP1:91,2] = PR[GP1:90,2] + 34.019;
   1:L PR[91] 10mm/sec CNT100;
   1:  PR[GP1:91,1] = PR[GP1:90,1] + 33.039;
   1:  PR[GP1:91,2] = PR[GP1:90,2] + 36.947;
   1:L PR[91] 10mm/sec CNT100;
   1:  PR[GP1:91,1] = PR[GP1:90,1] + 26.041;
   1:  PR[GP1:91,2] = PR[GP1:90,2] + 41.903;
   1:L PR[91] 10mm/sec CNT100;
   1:  PR[GP1:91,1] = PR[GP1:90,1] + 18.042;
   1:  PR[GP1:91,2] = PR[GP1:90,2] + 45.002;
   1:L PR[91] 10mm/sec CNT100;
   1:  PR[GP1:91,1] = PR[GP1:90,1] + 13.685;
   1:  PR[GP1:91,2] = PR[GP1:90,2] + 46.469;
   1:L PR[91] 10mm/sec CNT100;
   1:  PR[GP1:91,1] = PR[GP1:90,1] + 5.017;
   1:  PR[GP1:91,2] = PR[GP1:90,2] + 47.542;
   1:L PR[91] 10mm/sec CNT100;
   1:  PR[GP1:91,1] = PR[GP1:90,1] + 0.156;
   1:  PR[GP1:91,2] = PR[GP1:90,2] + 47.448;
   1:L PR[91] 10mm/sec CNT100;
   1:  PR[GP1:91,1] = PR[GP1:90,1] + -3.391;
   1:  PR[GP1:91,2] = PR[GP1:90,2] + 47.865;
   1:  PR[GP1:91,3] = PR[GP1:90,3] + 122.360;
   1:L PR[91] 10mm/sec CNT100;
   1:  PR[GP1:91,1] = PR[GP1:90,1] + -12.655;
   1:  PR[GP1:91,2] = PR[GP1:90,2] + 46.717;
   1:L PR[91] 10mm/sec CNT100;
   1:  PR[GP1:91,1] = PR[GP1:90,1] + -16.241;
   1:  PR[GP1:91,2] = PR[GP1:90,2] + 45.510;
   1:L PR[91] 10mm/sec CNT100;
   1:  PR[GP1:91,1] = PR[GP1:90,1] + -24.811;
   1:  PR[GP1:91,2] = PR[GP1:90,2] + 42.189;
   1:L PR[91] 10mm/sec CNT100;
   1:  PR[GP1:91,1] = PR[GP1:90,1] + -27.919;
   1:  PR[GP1:91,2] = PR[GP1:90,2] + 39.705;
   1:L PR[91] 10mm/sec CNT100;
   1:  PR[GP1:91,1] = PR[GP1:90,1] + -35.354;
   1:  PR[GP1:91,2] = PR[GP1:90,2] + 34.441;
   1:L PR[91] 10mm/sec CNT100;
   1:  PR[GP1:91,1] = PR[GP1:90,1] + -41.858;
   1:  PR[GP1:91,2] = PR[GP1:90,2] + 26.606;
   1:L PR[91] 10mm/sec CNT100;
   1:  PR[GP1:91,1] = PR[GP1:90,1] + -43.905;
   1:  PR[GP1:91,2] = PR[GP1:90,2] + 23.187;
   1:L PR[91] 10mm/sec CNT100;
   1:  PR[GP1:91,1] = PR[GP1:90,1] + -47.984;
   1:  PR[GP1:91,2] = PR[GP1:90,2] + 13.947;
   1:L PR[91] 10mm/sec CNT100;
   1:  PR[GP1:91,1] = PR[GP1:90,1] + -48.712;
   1:  PR[GP1:91,2] = PR[GP1:90,2] + 9.958;
   1:L PR[91] 10mm/sec CNT100;
   1:  PR[GP1:91,1] = PR[GP1:90,1] + -50.099;
   1:  PR[GP1:91,2] = PR[GP1:90,2] + 0.008;
   1:L PR[91] 10mm/sec CNT100;
   1:  PR[GP1:91,1] = PR[GP1:90,1] + -49.380;
   1:  PR[GP1:91,2] = PR[GP1:90,2] + -3.925;
   1:L PR[91] 10mm/sec CNT100;
   1:  PR[GP1:91,1] = PR[GP1:90,1] + -47.979;
   1:  PR[GP1:91,2] = PR[GP1:90,2] + -13.967;
   1:L PR[91] 10mm/sec CNT100;
   1:  PR[GP1:91,1] = PR[GP1:90,1] + -43.905;
   1:  PR[GP1:91,2] = PR[GP1:90,2] + -23.196;
   1:L PR[91] 10mm/sec CNT100;
   1:  PR[GP1:91,1] = PR[GP1:90,1] + -41.858;
   1:  PR[GP1:91,2] = PR[GP1:90,2] + -26.615;
   1:L PR[91] 10mm/sec CNT100;
   1:  PR[GP1:91,1] = PR[GP1:90,1] + -35.342;
   1:  PR[GP1:91,2] = PR[GP1:90,2] + -34.464;
   1:L PR[91] 10mm/sec CNT100;
   1:  PR[GP1:91,1] = PR[GP1:90,1] + -32.340;
   1:  PR[GP1:91,2] = PR[GP1:90,2] + -36.872;
   1:L PR[91] 10mm/sec CNT100;
   1:  PR[GP1:91,1] = PR[GP1:90,1] + -24.828;
   1:  PR[GP1:91,2] = PR[GP1:90,2] + -42.191;
   1:L PR[91] 10mm/sec CNT100;
   1:  PR[GP1:91,1] = PR[GP1:90,1] + -16.241;
   1:  PR[GP1:91,2] = PR[GP1:90,2] + -45.519;
   1:L PR[91] 10mm/sec CNT100;
   1:  PR[GP1:91,1] = PR[GP1:90,1] + -12.656;
   1:  PR[GP1:91,2] = PR[GP1:90,2] + -46.726;
   1:L PR[91] 10mm/sec CNT100;
   1:  PR[GP1:91,1] = PR[GP1:90,1] + -3.392;
   1:  PR[GP1:91,2] = PR[GP1:90,2] + -47.874;
   1:L PR[91] 10mm/sec CNT100;
   1:  PR[GP1:91,1] = PR[GP1:90,1] + 0.199;
   1:  PR[GP1:91,2] = PR[GP1:90,2] + -47.796;
   1:L PR[91] 10mm/sec CNT100;
   1:  PR[GP1:91,1] = PR[GP1:90,1] + 4.210;
   1:  PR[GP1:91,2] = PR[GP1:90,2] + -47.874;
   1:L PR[91] 10mm/sec CNT100;
   1:  PR[GP1:91,1] = PR[GP1:90,1] + 13.475;
   1:  PR[GP1:91,2] = PR[GP1:90,2] + -46.726;
   1:L PR[91] 10mm/sec CNT100;
   1:  PR[GP1:91,1] = PR[GP1:90,1] + 17.061;
   1:  PR[GP1:91,2] = PR[GP1:90,2] + -45.519;
   1:L PR[91] 10mm/sec CNT100;
   1:  PR[GP1:91,1] = PR[GP1:90,1] + 25.632;
   1:  PR[GP1:91,2] = PR[GP1:90,2] + -42.198;
   1:L PR[91] 10mm/sec CNT100;
   1:  PR[GP1:91,1] = PR[GP1:90,1] + 28.740;
   1:  PR[GP1:91,2] = PR[GP1:90,2] + -39.713;
   1:L PR[91] 10mm/sec CNT100;
   1:  PR[GP1:91,1] = PR[GP1:90,1] + 36.176;
   1:  PR[GP1:91,2] = PR[GP1:90,2] + -34.448;
   1:L PR[91] 10mm/sec CNT100;
   1:  PR[GP1:91,1] = PR[GP1:90,1] + 42.680;
   1:  PR[GP1:91,2] = PR[GP1:90,2] + -26.614;
   1:L PR[91] 10mm/sec CNT100;
   1:  PR[GP1:91,1] = PR[GP1:90,1] + 44.726;
   1:  PR[GP1:91,2] = PR[GP1:90,2] + -23.196;
   1:L PR[91] 10mm/sec CNT100;
   1:  PR[GP1:91,1] = PR[GP1:90,1] + 48.805;
   1:  PR[GP1:91,2] = PR[GP1:90,2] + -13.956;
   1:L PR[91] 10mm/sec CNT100;
   1:  PR[GP1:91,1] = PR[GP1:90,1] + 49.532;
   1:  PR[GP1:91,2] = PR[GP1:90,2] + -9.966;
   1:L PR[91] 10mm/sec CNT100;
   1:  PR[GP1:91,1] = PR[GP1:90,1] + 50.920;
   1:  PR[GP1:91,2] = PR[GP1:90,2] + -0.017;
   1:L PR[91] 10mm/sec CNT100;
   1:  PR[GP1:91,1] = PR[GP1:90,1] + 50.200;
   1:  PR[GP1:91,2] = PR[GP1:90,2] + 3.918;
   1:L PR[91] 10mm/sec CNT100;
   1:  PR[GP1:91,1] = PR[GP1:90,1] + 48.800;
   1:  PR[GP1:91,2] = PR[GP1:90,2] + 13.959;
   1:L PR[91] 10mm/sec CNT100;
   1:  PR[GP1:91,1] = PR[GP1:90,1] + 44.726;
   1:  PR[GP1:91,2] = PR[GP1:90,2] + 23.188;
   1:L PR[91] 10mm/sec CNT100;
   1:  PR[GP1:91,1] = PR[GP1:90,1] + 42.679;
   1:  PR[GP1:91,2] = PR[GP1:90,2] + 26.605;
   1:L PR[91] 10mm/sec CNT100;
   1:  PR[GP1:91,1] = PR[GP1:90,1] + 36.164;
   1:  PR[GP1:91,2] = PR[GP1:90,2] + 34.453;
   1:L PR[91] 10mm/sec CNT100;
   1:  PR[GP1:91,1] = PR[GP1:90,1] + 33.161;
   1:  PR[GP1:91,2] = PR[GP1:90,2] + 36.862;
   1:L PR[91] 10mm/sec CNT100;
   1:  PR[GP1:91,1] = PR[GP1:90,1] + 25.648;
   1:  PR[GP1:91,2] = PR[GP1:90,2] + 42.183;
   1:L PR[91] 10mm/sec CNT100;
   1:  PR[GP1:91,1] = PR[GP1:90,1] + 17.060;
   1:  PR[GP1:91,2] = PR[GP1:90,2] + 45.511;
   1:L PR[91] 10mm/sec CNT100;
   1:  PR[GP1:91,1] = PR[GP1:90,1] + 13.474;
   1:  PR[GP1:91,2] = PR[GP1:90,2] + 46.718;
   1:L PR[91] 10mm/sec CNT100;
   1:  PR[GP1:91,1] = PR[GP1:90,1] + 4.209;
   1:  PR[GP1:91,2] = PR[GP1:90,2] + 47.865;
   1:L PR[91] 10mm/sec CNT100;
   1:  PR[GP1:91,1] = PR[GP1:90,1] + 0.200;
   1:  PR[GP1:91,2] = PR[GP1:90,2] + 47.788;
   1:L PR[91] 10mm/sec CNT100;
   1:  PR[GP1:91,1] = PR[GP1:90,1] + -2.583;
   1:  PR[GP1:91,2] = PR[GP1:90,2] + 48.188;
   1:  PR[GP1:91,3] = PR[GP1:90,3] + 123.690;
   1:L PR[91] 10mm/sec CNT100;
   1:  PR[GP1:91,1] = PR[GP1:90,1] + -12.444;
   1:  PR[GP1:91,2] = PR[GP1:90,2] + 46.966;
   1:L PR[91] 10mm/sec CNT100;
   1:  PR[GP1:91,1] = PR[GP1:90,1] + -15.259;
   1:  PR[GP1:91,2] = PR[GP1:90,2] + 46.019;
   1:L PR[91] 10mm/sec CNT100;
   1:  PR[GP1:91,1] = PR[GP1:90,1] + -24.418;
   1:  PR[GP1:91,2] = PR[GP1:90,2] + 42.469;
   1:L PR[91] 10mm/sec CNT100;
   1:  PR[GP1:91,1] = PR[GP1:90,1] + -26.858;
   1:  PR[GP1:91,2] = PR[GP1:90,2] + 40.519;
   1:L PR[91] 10mm/sec CNT100;
   1:  PR[GP1:91,1] = PR[GP1:90,1] + -34.829;
   1:  PR[GP1:91,2] = PR[GP1:90,2] + 34.875;
   1:L PR[91] 10mm/sec CNT100;
   1:  PR[GP1:91,1] = PR[GP1:90,1] + -41.806;
   1:  PR[GP1:91,2] = PR[GP1:90,2] + 26.471;
   1:L PR[91] 10mm/sec CNT100;
   1:  PR[GP1:91,1] = PR[GP1:90,1] + -43.412;
   1:  PR[GP1:91,2] = PR[GP1:90,2] + 23.788;
   1:L PR[91] 10mm/sec CNT100;
   1:  PR[GP1:91,1] = PR[GP1:90,1] + -47.799;
   1:  PR[GP1:91,2] = PR[GP1:90,2] + 13.852;
   1:L PR[91] 10mm/sec CNT100;
   1:  PR[GP1:91,1] = PR[GP1:90,1] + -48.369;
   1:  PR[GP1:91,2] = PR[GP1:90,2] + 10.722;
   1:L PR[91] 10mm/sec CNT100;
   1:  PR[GP1:91,1] = PR[GP1:90,1] + -49.864;
   1:  PR[GP1:91,2] = PR[GP1:90,2] + 0.008;
   1:L PR[91] 10mm/sec CNT100;
   1:  PR[GP1:91,1] = PR[GP1:90,1] + -49.299;
   1:  PR[GP1:91,2] = PR[GP1:90,2] + -3.078;
   1:L PR[91] 10mm/sec CNT100;
   1:  PR[GP1:91,1] = PR[GP1:90,1] + -47.794;
   1:  PR[GP1:91,2] = PR[GP1:90,2] + -13.873;
   1:L PR[91] 10mm/sec CNT100;
   1:  PR[GP1:91,1] = PR[GP1:90,1] + -43.412;
   1:  PR[GP1:91,2] = PR[GP1:90,2] + -23.797;
   1:L PR[91] 10mm/sec CNT100;
   1:  PR[GP1:91,1] = PR[GP1:90,1] + -41.806;
   1:  PR[GP1:91,2] = PR[GP1:90,2] + -26.480;
   1:L PR[91] 10mm/sec CNT100;
   1:  PR[GP1:91,1] = PR[GP1:90,1] + -34.818;
   1:  PR[GP1:91,2] = PR[GP1:90,2] + -34.897;
   1:L PR[91] 10mm/sec CNT100;
   1:  PR[GP1:91,1] = PR[GP1:90,1] + -32.462;
   1:  PR[GP1:91,2] = PR[GP1:90,2] + -36.787;
   1:L PR[91] 10mm/sec CNT100;
   1:  PR[GP1:91,1] = PR[GP1:90,1] + -24.435;
   1:  PR[GP1:91,2] = PR[GP1:90,2] + -42.471;
   1:L PR[91] 10mm/sec CNT100;
   1:  PR[GP1:91,1] = PR[GP1:90,1] + -15.259;
   1:  PR[GP1:91,2] = PR[GP1:90,2] + -46.027;
   1:L PR[91] 10mm/sec CNT100;
   1:  PR[GP1:91,1] = PR[GP1:90,1] + -12.445;
   1:  PR[GP1:91,2] = PR[GP1:90,2] + -46.975;
   1:L PR[91] 10mm/sec CNT100;
   1:  PR[GP1:91,1] = PR[GP1:90,1] + -2.584;
   1:  PR[GP1:91,2] = PR[GP1:90,2] + -48.196;
   1:L PR[91] 10mm/sec CNT100;
   1:  PR[GP1:91,1] = PR[GP1:90,1] + 0.243;
   1:  PR[GP1:91,2] = PR[GP1:90,2] + -48.136;
   1:L PR[91] 10mm/sec CNT100;
   1:  PR[GP1:91,1] = PR[GP1:90,1] + 3.401;
   1:  PR[GP1:91,2] = PR[GP1:90,2] + -48.196;
   1:L PR[91] 10mm/sec CNT100;
   1:  PR[GP1:91,1] = PR[GP1:90,1] + 13.264;
   1:  PR[GP1:91,2] = PR[GP1:90,2] + -46.975;
   1:L PR[91] 10mm/sec CNT100;
   1:  PR[GP1:91,1] = PR[GP1:90,1] + 16.079;
   1:  PR[GP1:91,2] = PR[GP1:90,2] + -46.028;
   1:L PR[91] 10mm/sec CNT100;
   1:  PR[GP1:91,1] = PR[GP1:90,1] + 25.239;
   1:  PR[GP1:91,2] = PR[GP1:90,2] + -42.478;
   1:L PR[91] 10mm/sec CNT100;
   1:  PR[GP1:91,1] = PR[GP1:90,1] + 27.679;
   1:  PR[GP1:91,2] = PR[GP1:90,2] + -40.527;
   1:L PR[91] 10mm/sec CNT100;
   1:  PR[GP1:91,1] = PR[GP1:90,1] + 35.652;
   1:  PR[GP1:91,2] = PR[GP1:90,2] + -34.881;
   1:L PR[91] 10mm/sec CNT100;
   1:  PR[GP1:91,1] = PR[GP1:90,1] + 42.628;
   1:  PR[GP1:91,2] = PR[GP1:90,2] + -26.479;
   1:L PR[91] 10mm/sec CNT100;
   1:  PR[GP1:91,1] = PR[GP1:90,1] + 44.233;
   1:  PR[GP1:91,2] = PR[GP1:90,2] + -23.797;
   1:L PR[91] 10mm/sec CNT100;
   1:  PR[GP1:91,1] = PR[GP1:90,1] + 48.619;
   1:  PR[GP1:91,2] = PR[GP1:90,2] + -13.862;
   1:L PR[91] 10mm/sec CNT100;
   1:  PR[GP1:91,1] = PR[GP1:90,1] + 49.190;
   1:  PR[GP1:91,2] = PR[GP1:90,2] + -10.731;
   1:L PR[91] 10mm/sec CNT100;
   1:  PR[GP1:91,1] = PR[GP1:90,1] + 50.684;
   1:  PR[GP1:91,2] = PR[GP1:90,2] + -0.017;
   1:L PR[91] 10mm/sec CNT100;
   1:  PR[GP1:91,1] = PR[GP1:90,1] + 50.120;
   1:  PR[GP1:91,2] = PR[GP1:90,2] + 3.070;
   1:L PR[91] 10mm/sec CNT100;
   1:  PR[GP1:91,1] = PR[GP1:90,1] + 48.614;
   1:  PR[GP1:91,2] = PR[GP1:90,2] + 13.865;
   1:L PR[91] 10mm/sec CNT100;
   1:  PR[GP1:91,1] = PR[GP1:90,1] + 44.233;
   1:  PR[GP1:91,2] = PR[GP1:90,2] + 23.789;
   1:L PR[91] 10mm/sec CNT100;
   1:  PR[GP1:91,1] = PR[GP1:90,1] + 42.627;
   1:  PR[GP1:91,2] = PR[GP1:90,2] + 26.470;
   1:L PR[91] 10mm/sec CNT100;
   1:  PR[GP1:91,1] = PR[GP1:90,1] + 35.640;
   1:  PR[GP1:91,2] = PR[GP1:90,2] + 34.887;
   1:L PR[91] 10mm/sec CNT100;
   1:  PR[GP1:91,1] = PR[GP1:90,1] + 33.284;
   1:  PR[GP1:91,2] = PR[GP1:90,2] + 36.778;
   1:L PR[91] 10mm/sec CNT100;
   1:  PR[GP1:91,1] = PR[GP1:90,1] + 25.255;
   1:  PR[GP1:91,2] = PR[GP1:90,2] + 42.463;
   1:L PR[91] 10mm/sec CNT100;
   1:  PR[GP1:91,1] = PR[GP1:90,1] + 16.078;
   1:  PR[GP1:91,2] = PR[GP1:90,2] + 46.019;
   1:L PR[91] 10mm/sec CNT100;
   1:  PR[GP1:91,1] = PR[GP1:90,1] + 13.263;
   1:  PR[GP1:91,2] = PR[GP1:90,2] + 46.966;
   1:L PR[91] 10mm/sec CNT100;
   1:  PR[GP1:91,1] = PR[GP1:90,1] + 3.400;
   1:  PR[GP1:91,2] = PR[GP1:90,2] + 48.188;
   1:L PR[91] 10mm/sec CNT100;
   1:  PR[GP1:91,1] = PR[GP1:90,1] + 0.244;
   1:  PR[GP1:91,2] = PR[GP1:90,2] + 48.127;
   1:L PR[91] 10mm/sec CNT100;
   1:  PR[GP1:91,1] = PR[GP1:90,1] + -1.775;
   1:  PR[GP1:91,2] = PR[GP1:90,2] + 48.510;
   1:  PR[GP1:91,3] = PR[GP1:90,3] + 125.020;
   1:L PR[91] 10mm/sec CNT100;
   1:  PR[GP1:91,1] = PR[GP1:90,1] + -12.234;
   1:  PR[GP1:91,2] = PR[GP1:90,2] + 47.215;
   1:L PR[91] 10mm/sec CNT100;
   1:  PR[GP1:91,1] = PR[GP1:90,1] + -14.277;
   1:  PR[GP1:91,2] = PR[GP1:90,2] + 46.527;
   1:L PR[91] 10mm/sec CNT100;
   1:  PR[GP1:91,1] = PR[GP1:90,1] + -24.025;
   1:  PR[GP1:91,2] = PR[GP1:90,2] + 42.749;
   1:L PR[91] 10mm/sec CNT100;
   1:  PR[GP1:91,1] = PR[GP1:90,1] + -25.797;
   1:  PR[GP1:91,2] = PR[GP1:90,2] + 41.333;
   1:L PR[91] 10mm/sec CNT100;
   1:  PR[GP1:91,1] = PR[GP1:90,1] + -34.305;
   1:  PR[GP1:91,2] = PR[GP1:90,2] + 35.309;
   1:L PR[91] 10mm/sec CNT100;
   1:  PR[GP1:91,1] = PR[GP1:90,1] + -41.754;
   1:  PR[GP1:91,2] = PR[GP1:90,2] + 26.336;
   1:L PR[91] 10mm/sec CNT100;
   1:  PR[GP1:91,1] = PR[GP1:90,1] + -42.919;
   1:  PR[GP1:91,2] = PR[GP1:90,2] + 24.390;
   1:L PR[91] 10mm/sec CNT100;
   1:  PR[GP1:91,1] = PR[GP1:90,1] + -47.613;
   1:  PR[GP1:91,2] = PR[GP1:90,2] + 13.758;
   1:L PR[91] 10mm/sec CNT100;
   1:  PR[GP1:91,1] = PR[GP1:90,1] + -48.027;
   1:  PR[GP1:91,2] = PR[GP1:90,2] + 11.487;
   1:L PR[91] 10mm/sec CNT100;
   1:  PR[GP1:91,1] = PR[GP1:90,1] + -49.628;
   1:  PR[GP1:91,2] = PR[GP1:90,2] + 0.008;
   1:L PR[91] 10mm/sec CNT100;
   1:  PR[GP1:91,1] = PR[GP1:90,1] + -49.218;
   1:  PR[GP1:91,2] = PR[GP1:90,2] + -2.231;
   1:L PR[91] 10mm/sec CNT100;
   1:  PR[GP1:91,1] = PR[GP1:90,1] + -47.608;
   1:  PR[GP1:91,2] = PR[GP1:90,2] + -13.778;
   1:L PR[91] 10mm/sec CNT100;
   1:  PR[GP1:91,1] = PR[GP1:90,1] + -42.919;
   1:  PR[GP1:91,2] = PR[GP1:90,2] + -24.398;
   1:L PR[91] 10mm/sec CNT100;
   1:  PR[GP1:91,1] = PR[GP1:90,1] + -41.754;
   1:  PR[GP1:91,2] = PR[GP1:90,2] + -26.345;
   1:L PR[91] 10mm/sec CNT100;
   1:  PR[GP1:91,1] = PR[GP1:90,1] + -34.294;
   1:  PR[GP1:91,2] = PR[GP1:90,2] + -35.331;
   1:L PR[91] 10mm/sec CNT100;
   1:  PR[GP1:91,1] = PR[GP1:90,1] + -32.584;
   1:  PR[GP1:91,2] = PR[GP1:90,2] + -36.702;
   1:L PR[91] 10mm/sec CNT100;
   1:  PR[GP1:91,1] = PR[GP1:90,1] + -24.042;
   1:  PR[GP1:91,2] = PR[GP1:90,2] + -42.752;
   1:L PR[91] 10mm/sec CNT100;
   1:  PR[GP1:91,1] = PR[GP1:90,1] + -14.277;
   1:  PR[GP1:91,2] = PR[GP1:90,2] + -46.536;
   1:L PR[91] 10mm/sec CNT100;
   1:  PR[GP1:91,1] = PR[GP1:90,1] + -12.234;
   1:  PR[GP1:91,2] = PR[GP1:90,2] + -47.223;
   1:L PR[91] 10mm/sec CNT100;
   1:  PR[GP1:91,1] = PR[GP1:90,1] + -1.776;
   1:  PR[GP1:91,2] = PR[GP1:90,2] + -48.519;
   1:L PR[91] 10mm/sec CNT100;
   1:  PR[GP1:91,1] = PR[GP1:90,1] + 0.287;
   1:  PR[GP1:91,2] = PR[GP1:90,2] + -48.475;
   1:L PR[91] 10mm/sec CNT100;
   1:  PR[GP1:91,1] = PR[GP1:90,1] + 2.593;
   1:  PR[GP1:91,2] = PR[GP1:90,2] + -48.519;
   1:L PR[91] 10mm/sec CNT100;
   1:  PR[GP1:91,1] = PR[GP1:90,1] + 13.053;
   1:  PR[GP1:91,2] = PR[GP1:90,2] + -47.224;
   1:L PR[91] 10mm/sec CNT100;
   1:  PR[GP1:91,1] = PR[GP1:90,1] + 15.096;
   1:  PR[GP1:91,2] = PR[GP1:90,2] + -46.536;
   1:L PR[91] 10mm/sec CNT100;
   1:  PR[GP1:91,1] = PR[GP1:90,1] + 24.846;
   1:  PR[GP1:91,2] = PR[GP1:90,2] + -42.758;
   1:L PR[91] 10mm/sec CNT100;
   1:  PR[GP1:91,1] = PR[GP1:90,1] + 26.618;
   1:  PR[GP1:91,2] = PR[GP1:90,2] + -41.342;
   1:L PR[91] 10mm/sec CNT100;
   1:  PR[GP1:91,1] = PR[GP1:90,1] + 35.128;
   1:  PR[GP1:91,2] = PR[GP1:90,2] + -35.315;
   1:L PR[91] 10mm/sec CNT100;
   1:  PR[GP1:91,1] = PR[GP1:90,1] + 42.576;
   1:  PR[GP1:91,2] = PR[GP1:90,2] + -26.344;
   1:L PR[91] 10mm/sec CNT100;
   1:  PR[GP1:91,1] = PR[GP1:90,1] + 43.741;
   1:  PR[GP1:91,2] = PR[GP1:90,2] + -24.398;
   1:L PR[91] 10mm/sec CNT100;
   1:  PR[GP1:91,1] = PR[GP1:90,1] + 48.434;
   1:  PR[GP1:91,2] = PR[GP1:90,2] + -13.767;
   1:L PR[91] 10mm/sec CNT100;
   1:  PR[GP1:91,1] = PR[GP1:90,1] + 48.848;
   1:  PR[GP1:91,2] = PR[GP1:90,2] + -11.495;
   1:L PR[91] 10mm/sec CNT100;
   1:  PR[GP1:91,1] = PR[GP1:90,1] + 50.449;
   1:  PR[GP1:91,2] = PR[GP1:90,2] + -0.017;
   1:L PR[91] 10mm/sec CNT100;
   1:  PR[GP1:91,1] = PR[GP1:90,1] + 50.039;
   1:  PR[GP1:91,2] = PR[GP1:90,2] + 2.223;
   1:L PR[91] 10mm/sec CNT100;
   1:  PR[GP1:91,1] = PR[GP1:90,1] + 48.429;
   1:  PR[GP1:91,2] = PR[GP1:90,2] + 13.770;
   1:L PR[91] 10mm/sec CNT100;
   1:  PR[GP1:91,1] = PR[GP1:90,1] + 43.741;
   1:  PR[GP1:91,2] = PR[GP1:90,2] + 24.389;
   1:L PR[91] 10mm/sec CNT100;
   1:  PR[GP1:91,1] = PR[GP1:90,1] + 42.575;
   1:  PR[GP1:91,2] = PR[GP1:90,2] + 26.335;
   1:L PR[91] 10mm/sec CNT100;
   1:  PR[GP1:91,1] = PR[GP1:90,1] + 35.116;
   1:  PR[GP1:91,2] = PR[GP1:90,2] + 35.321;
   1:L PR[91] 10mm/sec CNT100;
   1:  PR[GP1:91,1] = PR[GP1:90,1] + 33.406;
   1:  PR[GP1:91,2] = PR[GP1:90,2] + 36.693;
   1:L PR[91] 10mm/sec CNT100;
   1:  PR[GP1:91,1] = PR[GP1:90,1] + 24.862;
   1:  PR[GP1:91,2] = PR[GP1:90,2] + 42.743;
   1:L PR[91] 10mm/sec CNT100;
   1:  PR[GP1:91,1] = PR[GP1:90,1] + 15.096;
   1:  PR[GP1:91,2] = PR[GP1:90,2] + 46.527;
   1:L PR[91] 10mm/sec CNT100;
   1:  PR[GP1:91,1] = PR[GP1:90,1] + 13.053;
   1:  PR[GP1:91,2] = PR[GP1:90,2] + 47.215;
   1:L PR[91] 10mm/sec CNT100;
   1:  PR[GP1:91,1] = PR[GP1:90,1] + 2.592;
   1:  PR[GP1:91,2] = PR[GP1:90,2] + 48.510;
   1:L PR[91] 10mm/sec CNT100;
   1:  PR[GP1:91,1] = PR[GP1:90,1] + 0.287;
   1:  PR[GP1:91,2] = PR[GP1:90,2] + 48.466;
   1:L PR[91] 10mm/sec CNT100;
   1:  PR[GP1:91,1] = PR[GP1:90,1] + -0.967;
   1:  PR[GP1:91,2] = PR[GP1:90,2] + 48.833;
   1:  PR[GP1:91,3] = PR[GP1:90,3] + 126.350;
   1:L PR[91] 10mm/sec CNT100;
   1:  PR[GP1:91,1] = PR[GP1:90,1] + -12.023;
   1:  PR[GP1:91,2] = PR[GP1:90,2] + 47.463;
   1:L PR[91] 10mm/sec CNT100;
   1:  PR[GP1:91,1] = PR[GP1:90,1] + -13.295;
   1:  PR[GP1:91,2] = PR[GP1:90,2] + 47.035;
   1:L PR[91] 10mm/sec CNT100;
   1:  PR[GP1:91,1] = PR[GP1:90,1] + -23.632;
   1:  PR[GP1:91,2] = PR[GP1:90,2] + 43.029;
   1:L PR[91] 10mm/sec CNT100;
   1:  PR[GP1:91,1] = PR[GP1:90,1] + -24.736;
   1:  PR[GP1:91,2] = PR[GP1:90,2] + 42.147;
   1:L PR[91] 10mm/sec CNT100;
   1:  PR[GP1:91,1] = PR[GP1:90,1] + -33.781;
   1:  PR[GP1:91,2] = PR[GP1:90,2] + 35.742;
   1:L PR[91] 10mm/sec CNT100;
   1:  PR[GP1:91,1] = PR[GP1:90,1] + -41.702;
   1:  PR[GP1:91,2] = PR[GP1:90,2] + 26.201;
   1:L PR[91] 10mm/sec CNT100;
   1:  PR[GP1:91,1] = PR[GP1:90,1] + -42.427;
   1:  PR[GP1:91,2] = PR[GP1:90,2] + 24.991;
   1:L PR[91] 10mm/sec CNT100;
   1:  PR[GP1:91,1] = PR[GP1:90,1] + -47.427;
   1:  PR[GP1:91,2] = PR[GP1:90,2] + 13.664;
   1:L PR[91] 10mm/sec CNT100;
   1:  PR[GP1:91,1] = PR[GP1:90,1] + -47.685;
   1:  PR[GP1:91,2] = PR[GP1:90,2] + 12.251;
   1:L PR[91] 10mm/sec CNT100;
   1:  PR[GP1:91,1] = PR[GP1:90,1] + -49.392;
   1:  PR[GP1:91,2] = PR[GP1:90,2] + 0.008;
   1:L PR[91] 10mm/sec CNT100;
   1:  PR[GP1:91,1] = PR[GP1:90,1] + -49.138;
   1:  PR[GP1:91,2] = PR[GP1:90,2] + -1.384;
   1:L PR[91] 10mm/sec CNT100;
   1:  PR[GP1:91,1] = PR[GP1:90,1] + -47.422;
   1:  PR[GP1:91,2] = PR[GP1:90,2] + -13.684;
   1:L PR[91] 10mm/sec CNT100;
   1:  PR[GP1:91,1] = PR[GP1:90,1] + -42.427;
   1:  PR[GP1:91,2] = PR[GP1:90,2] + -24.999;
   1:L PR[91] 10mm/sec CNT100;
   1:  PR[GP1:91,1] = PR[GP1:90,1] + -41.702;
   1:  PR[GP1:91,2] = PR[GP1:90,2] + -26.210;
   1:L PR[91] 10mm/sec CNT100;
   1:  PR[GP1:91,1] = PR[GP1:90,1] + -33.769;
   1:  PR[GP1:91,2] = PR[GP1:90,2] + -35.765;
   1:L PR[91] 10mm/sec CNT100;
   1:  PR[GP1:91,1] = PR[GP1:90,1] + -32.706;
   1:  PR[GP1:91,2] = PR[GP1:90,2] + -36.618;
   1:L PR[91] 10mm/sec CNT100;
   1:  PR[GP1:91,1] = PR[GP1:90,1] + -23.648;
   1:  PR[GP1:91,2] = PR[GP1:90,2] + -43.032;
   1:L PR[91] 10mm/sec CNT100;
   1:  PR[GP1:91,1] = PR[GP1:90,1] + -13.295;
   1:  PR[GP1:91,2] = PR[GP1:90,2] + -47.044;
   1:L PR[91] 10mm/sec CNT100;
   1:  PR[GP1:91,1] = PR[GP1:90,1] + -12.023;
   1:  PR[GP1:91,2] = PR[GP1:90,2] + -47.472;
   1:L PR[91] 10mm/sec CNT100;
   1:  PR[GP1:91,1] = PR[GP1:90,1] + -0.968;
   1:  PR[GP1:91,2] = PR[GP1:90,2] + -48.842;
   1:L PR[91] 10mm/sec CNT100;
   1:  PR[GP1:91,1] = PR[GP1:90,1] + 0.331;
   1:  PR[GP1:91,2] = PR[GP1:90,2] + -48.814;
   1:L PR[91] 10mm/sec CNT100;
   1:  PR[GP1:91,1] = PR[GP1:90,1] + 1.784;
   1:  PR[GP1:91,2] = PR[GP1:90,2] + -48.842;
   1:L PR[91] 10mm/sec CNT100;
   1:  PR[GP1:91,1] = PR[GP1:90,1] + 12.842;
   1:  PR[GP1:91,2] = PR[GP1:90,2] + -47.473;
   1:L PR[91] 10mm/sec CNT100;
   1:  PR[GP1:91,1] = PR[GP1:90,1] + 14.114;
   1:  PR[GP1:91,2] = PR[GP1:90,2] + -47.044;
   1:L PR[91] 10mm/sec CNT100;
   1:  PR[GP1:91,1] = PR[GP1:90,1] + 24.452;
   1:  PR[GP1:91,2] = PR[GP1:90,2] + -43.038;
   1:L PR[91] 10mm/sec CNT100;
   1:  PR[GP1:91,1] = PR[GP1:90,1] + 25.556;
   1:  PR[GP1:91,2] = PR[GP1:90,2] + -42.156;
   1:L PR[91] 10mm/sec CNT100;
   1:  PR[GP1:91,1] = PR[GP1:90,1] + 34.604;
   1:  PR[GP1:91,2] = PR[GP1:90,2] + -35.749;
   1:L PR[91] 10mm/sec CNT100;
   1:  PR[GP1:91,1] = PR[GP1:90,1] + 42.523;
   1:  PR[GP1:91,2] = PR[GP1:90,2] + -26.209;
   1:L PR[91] 10mm/sec CNT100;
   1:  PR[GP1:91,1] = PR[GP1:90,1] + 43.248;
   1:  PR[GP1:91,2] = PR[GP1:90,2] + -24.999;
   1:L PR[91] 10mm/sec CNT100;
   1:  PR[GP1:91,1] = PR[GP1:90,1] + 48.248;
   1:  PR[GP1:91,2] = PR[GP1:90,2] + -13.673;
   1:L PR[91] 10mm/sec CNT100;
   1:  PR[GP1:91,1] = PR[GP1:90,1] + 48.505;
   1:  PR[GP1:91,2] = PR[GP1:90,2] + -12.260;
   1:L PR[91] 10mm/sec CNT100;
   1:  PR[GP1:91,1] = PR[GP1:90,1] + 50.213;
   1:  PR[GP1:91,2] = PR[GP1:90,2] + -0.017;
   1:L PR[91] 10mm/sec CNT100;
   1:  PR[GP1:91,1] = PR[GP1:90,1] + 49.958;
   1:  PR[GP1:91,2] = PR[GP1:90,2] + 1.375;
   1:L PR[91] 10mm/sec CNT100;
   1:  PR[GP1:91,1] = PR[GP1:90,1] + 48.243;
   1:  PR[GP1:91,2] = PR[GP1:90,2] + 13.676;
   1:L PR[91] 10mm/sec CNT100;
   1:  PR[GP1:91,1] = PR[GP1:90,1] + 43.248;
   1:  PR[GP1:91,2] = PR[GP1:90,2] + 24.990;
   1:L PR[91] 10mm/sec CNT100;
   1:  PR[GP1:91,1] = PR[GP1:90,1] + 42.523;
   1:  PR[GP1:91,2] = PR[GP1:90,2] + 26.200;
   1:L PR[91] 10mm/sec CNT100;
   1:  PR[GP1:91,1] = PR[GP1:90,1] + 34.592;
   1:  PR[GP1:91,2] = PR[GP1:90,2] + 35.755;
   1:L PR[91] 10mm/sec CNT100;
   1:  PR[GP1:91,1] = PR[GP1:90,1] + 33.528;
   1:  PR[GP1:91,2] = PR[GP1:90,2] + 36.608;
   1:L PR[91] 10mm/sec CNT100;
   1:  PR[GP1:91,1] = PR[GP1:90,1] + 24.468;
   1:  PR[GP1:91,2] = PR[GP1:90,2] + 43.023;
   1:L PR[91] 10mm/sec CNT100;
   1:  PR[GP1:91,1] = PR[GP1:90,1] + 14.114;
   1:  PR[GP1:91,2] = PR[GP1:90,2] + 47.036;
   1:L PR[91] 10mm/sec CNT100;
   1:  PR[GP1:91,1] = PR[GP1:90,1] + 12.842;
   1:  PR[GP1:91,2] = PR[GP1:90,2] + 47.464;
   1:L PR[91] 10mm/sec CNT100;
   1:  PR[GP1:91,1] = PR[GP1:90,1] + 1.784;
   1:  PR[GP1:91,2] = PR[GP1:90,2] + 48.833;
   1:L PR[91] 10mm/sec CNT100;
   1:  PR[GP1:91,1] = PR[GP1:90,1] + 0.331;
   1:  PR[GP1:91,2] = PR[GP1:90,2] + 48.805;
   1:L PR[91] 10mm/sec CNT100;
   1:  PR[GP1:91,1] = PR[GP1:90,1] + -0.159;
   1:  PR[GP1:91,2] = PR[GP1:90,2] + 49.156;
   1:  PR[GP1:91,3] = PR[GP1:90,3] + 127.680;
   1:L PR[91] 10mm/sec CNT100;
   1:  PR[GP1:91,1] = PR[GP1:90,1] + -11.812;
   1:  PR[GP1:91,2] = PR[GP1:90,2] + 47.712;
   1:L PR[91] 10mm/sec CNT100;
   1:  PR[GP1:91,1] = PR[GP1:90,1] + -12.313;
   1:  PR[GP1:91,2] = PR[GP1:90,2] + 47.543;
   1:L PR[91] 10mm/sec CNT100;
   1:  PR[GP1:91,1] = PR[GP1:90,1] + -23.238;
   1:  PR[GP1:91,2] = PR[GP1:90,2] + 43.309;
   1:L PR[91] 10mm/sec CNT100;
   1:  PR[GP1:91,1] = PR[GP1:90,1] + -23.675;
   1:  PR[GP1:91,2] = PR[GP1:90,2] + 42.961;
   1:L PR[91] 10mm/sec CNT100;
   1:  PR[GP1:91,1] = PR[GP1:90,1] + -33.257;
   1:  PR[GP1:91,2] = PR[GP1:90,2] + 36.176;
   1:L PR[91] 10mm/sec CNT100;
   1:  PR[GP1:91,1] = PR[GP1:90,1] + -41.650;
   1:  PR[GP1:91,2] = PR[GP1:90,2] + 26.066;
   1:L PR[91] 10mm/sec CNT100;
   1:  PR[GP1:91,1] = PR[GP1:90,1] + -41.934;
   1:  PR[GP1:91,2] = PR[GP1:90,2] + 25.592;
   1:L PR[91] 10mm/sec CNT100;
   1:  PR[GP1:91,1] = PR[GP1:90,1] + -47.241;
   1:  PR[GP1:91,2] = PR[GP1:90,2] + 13.570;
   1:L PR[91] 10mm/sec CNT100;
   1:  PR[GP1:91,1] = PR[GP1:90,1] + -47.342;
   1:  PR[GP1:91,2] = PR[GP1:90,2] + 13.016;
   1:L PR[91] 10mm/sec CNT100;
   1:  PR[GP1:91,1] = PR[GP1:90,1] + -49.157;
   1:  PR[GP1:91,2] = PR[GP1:90,2] + 0.008;
   1:L PR[91] 10mm/sec CNT100;
   1:  PR[GP1:91,1] = PR[GP1:90,1] + -49.057;
   1:  PR[GP1:91,2] = PR[GP1:90,2] + -0.537;
   1:L PR[91] 10mm/sec CNT100;
   1:  PR[GP1:91,1] = PR[GP1:90,1] + -47.236;
   1:  PR[GP1:91,2] = PR[GP1:90,2] + -13.590;
   1:L PR[91] 10mm/sec CNT100;
   1:  PR[GP1:91,1] = PR[GP1:90,1] + -41.934;
   1:  PR[GP1:91,2] = PR[GP1:90,2] + -25.601;
   1:L PR[91] 10mm/sec CNT100;
   1:  PR[GP1:91,1] = PR[GP1:90,1] + -41.650;
   1:  PR[GP1:91,2] = PR[GP1:90,2] + -26.075;
   1:L PR[91] 10mm/sec CNT100;
   1:  PR[GP1:91,1] = PR[GP1:90,1] + -33.245;
   1:  PR[GP1:91,2] = PR[GP1:90,2] + -36.199;
   1:L PR[91] 10mm/sec CNT100;
   1:  PR[GP1:91,1] = PR[GP1:90,1] + -32.829;
   1:  PR[GP1:91,2] = PR[GP1:90,2] + -36.533;
   1:L PR[91] 10mm/sec CNT100;
   1:  PR[GP1:91,1] = PR[GP1:90,1] + -23.255;
   1:  PR[GP1:91,2] = PR[GP1:90,2] + -43.312;
   1:L PR[91] 10mm/sec CNT100;
   1:  PR[GP1:91,1] = PR[GP1:90,1] + -12.313;
   1:  PR[GP1:91,2] = PR[GP1:90,2] + -47.552;
   1:L PR[91] 10mm/sec CNT100;
   1:  PR[GP1:91,1] = PR[GP1:90,1] + -11.813;
   1:  PR[GP1:91,2] = PR[GP1:90,2] + -47.721;
   1:L PR[91] 10mm/sec CNT100;
   1:  PR[GP1:91,1] = PR[GP1:90,1] + -0.160;
   1:  PR[GP1:91,2] = PR[GP1:90,2] + -49.165;
   1:L PR[91] 10mm/sec CNT100;
   1:  PR[GP1:91,1] = PR[GP1:90,1] + 0.375;
   1:  PR[GP1:91,2] = PR[GP1:90,2] + -49.153;
   1:L PR[91] 10mm/sec CNT100;
   1:  PR[GP1:91,1] = PR[GP1:90,1] + 0.976;
   1:  PR[GP1:91,2] = PR[GP1:90,2] + -49.165;
   1:L PR[91] 10mm/sec CNT100;
   1:  PR[GP1:91,1] = PR[GP1:90,1] + 12.631;
   1:  PR[GP1:91,2] = PR[GP1:90,2] + -47.721;
   1:L PR[91] 10mm/sec CNT100;
   1:  PR[GP1:91,1] = PR[GP1:90,1] + 13.132;
   1:  PR[GP1:91,2] = PR[GP1:90,2] + -47.553;
   1:L PR[91] 10mm/sec CNT100;
   1:  PR[GP1:91,1] = PR[GP1:90,1] + 24.059;
   1:  PR[GP1:91,2] = PR[GP1:90,2] + -43.319;
   1:L PR[91] 10mm/sec CNT100;
   1:  PR[GP1:91,1] = PR[GP1:90,1] + 24.495;
   1:  PR[GP1:91,2] = PR[GP1:90,2] + -42.970;
   1:L PR[91] 10mm/sec CNT100;
   1:  PR[GP1:91,1] = PR[GP1:90,1] + 34.079;
   1:  PR[GP1:91,2] = PR[GP1:90,2] + -36.183;
   1:L PR[91] 10mm/sec CNT100;
   1:  PR[GP1:91,1] = PR[GP1:90,1] + 42.471;
   1:  PR[GP1:91,2] = PR[GP1:90,2] + -26.074;
   1:L PR[91] 10mm/sec CNT100;
   1:  PR[GP1:91,1] = PR[GP1:90,1] + 42.755;
   1:  PR[GP1:91,2] = PR[GP1:90,2] + -25.600;
   1:L PR[91] 10mm/sec CNT100;
   1:  PR[GP1:91,1] = PR[GP1:90,1] + 48.062;
   1:  PR[GP1:91,2] = PR[GP1:90,2] + -13.578;
   1:L PR[91] 10mm/sec CNT100;
   1:  PR[GP1:91,1] = PR[GP1:90,1] + 48.163;
   1:  PR[GP1:91,2] = PR[GP1:90,2] + -13.024;
   1:L PR[91] 10mm/sec CNT100;
   1:  PR[GP1:91,1] = PR[GP1:90,1] + 49.977;
   1:  PR[GP1:91,2] = PR[GP1:90,2] + -0.017;
   1:L PR[91] 10mm/sec CNT100;
   1:  PR[GP1:91,1] = PR[GP1:90,1] + 49.878;
   1:  PR[GP1:91,2] = PR[GP1:90,2] + 0.528;
   1:L PR[91] 10mm/sec CNT100;
   1:  PR[GP1:91,1] = PR[GP1:90,1] + 48.057;
   1:  PR[GP1:91,2] = PR[GP1:90,2] + 13.581;
   1:L PR[91] 10mm/sec CNT100;
   1:  PR[GP1:91,1] = PR[GP1:90,1] + 42.755;
   1:  PR[GP1:91,2] = PR[GP1:90,2] + 25.591;
   1:L PR[91] 10mm/sec CNT100;
   1:  PR[GP1:91,1] = PR[GP1:90,1] + 42.471;
   1:  PR[GP1:91,2] = PR[GP1:90,2] + 26.065;
   1:L PR[91] 10mm/sec CNT100;
   1:  PR[GP1:91,1] = PR[GP1:90,1] + 34.068;
   1:  PR[GP1:91,2] = PR[GP1:90,2] + 36.188;
   1:L PR[91] 10mm/sec CNT100;
   1:  PR[GP1:91,1] = PR[GP1:90,1] + 33.650;
   1:  PR[GP1:91,2] = PR[GP1:90,2] + 36.523;
   1:L PR[91] 10mm/sec CNT100;
   1:  PR[GP1:91,1] = PR[GP1:90,1] + 24.075;
   1:  PR[GP1:91,2] = PR[GP1:90,2] + 43.303;
   1:L PR[91] 10mm/sec CNT100;
   1:  PR[GP1:91,1] = PR[GP1:90,1] + 13.132;
   1:  PR[GP1:91,2] = PR[GP1:90,2] + 47.544;
   1:L PR[91] 10mm/sec CNT100;
   1:  PR[GP1:91,1] = PR[GP1:90,1] + 12.631;
   1:  PR[GP1:91,2] = PR[GP1:90,2] + 47.712;
   1:L PR[91] 10mm/sec CNT100;
   1:  PR[GP1:91,1] = PR[GP1:90,1] + 0.976;
   1:  PR[GP1:91,2] = PR[GP1:90,2] + 49.156;
   1:L PR[91] 10mm/sec CNT100;
   1:  PR[GP1:91,1] = PR[GP1:90,1] + 0.375;
   1:  PR[GP1:91,2] = PR[GP1:90,2] + 49.144;
   1:L PR[91] 10mm/sec CNT100;
   1:  PR[GP1:91,1] = PR[GP1:90,1] + -11.286;
   1:  PR[GP1:91,2] = PR[GP1:90,2] + 47.942;
   1:  PR[GP1:91,3] = PR[GP1:90,3] + 129.010;
   1:L PR[91] 10mm/sec CNT100;
   1:  PR[GP1:91,1] = PR[GP1:90,1] + -11.745;
   1:  PR[GP1:91,2] = PR[GP1:90,2] + 47.869;
   1:L PR[91] 10mm/sec CNT100;
   1:  PR[GP1:91,1] = PR[GP1:90,1] + -22.721;
   1:  PR[GP1:91,2] = PR[GP1:90,2] + 43.616;
   1:L PR[91] 10mm/sec CNT100;
   1:  PR[GP1:91,1] = PR[GP1:90,1] + -23.136;
   1:  PR[GP1:91,2] = PR[GP1:90,2] + 43.404;
   1:L PR[91] 10mm/sec CNT100;
   1:  PR[GP1:91,1] = PR[GP1:90,1] + -32.743;
   1:  PR[GP1:91,2] = PR[GP1:90,2] + 36.602;
   1:L PR[91] 10mm/sec CNT100;
   1:  PR[GP1:91,1] = PR[GP1:90,1] + -33.071;
   1:  PR[GP1:91,2] = PR[GP1:90,2] + 36.274;
   1:L PR[91] 10mm/sec CNT100;
   1:  PR[GP1:91,1] = PR[GP1:90,1] + -41.527;
   1:  PR[GP1:91,2] = PR[GP1:90,2] + 26.088;
   1:L PR[91] 10mm/sec CNT100;
   1:  PR[GP1:91,1] = PR[GP1:90,1] + -41.734;
   1:  PR[GP1:91,2] = PR[GP1:90,2] + 25.681;
   1:L PR[91] 10mm/sec CNT100;
   1:  PR[GP1:91,1] = PR[GP1:90,1] + -47.080;
   1:  PR[GP1:91,2] = PR[GP1:90,2] + 13.572;
   1:L PR[91] 10mm/sec CNT100;
   1:  PR[GP1:91,1] = PR[GP1:90,1] + -48.984;
   1:  PR[GP1:91,2] = PR[GP1:90,2] + -0.005;
   1:L PR[91] 10mm/sec CNT100;
   1:  PR[GP1:91,1] = PR[GP1:90,1] + -47.154;
   1:  PR[GP1:91,2] = PR[GP1:90,2] + -13.126;
   1:L PR[91] 10mm/sec CNT100;
   1:  PR[GP1:91,1] = PR[GP1:90,1] + -47.082;
   1:  PR[GP1:91,2] = PR[GP1:90,2] + -13.576;
   1:L PR[91] 10mm/sec CNT100;
   1:  PR[GP1:91,1] = PR[GP1:90,1] + -41.734;
   1:  PR[GP1:91,2] = PR[GP1:90,2] + -25.690;
   1:L PR[91] 10mm/sec CNT100;
   1:  PR[GP1:91,1] = PR[GP1:90,1] + -41.527;
   1:  PR[GP1:91,2] = PR[GP1:90,2] + -26.096;
   1:L PR[91] 10mm/sec CNT100;
   1:  PR[GP1:91,1] = PR[GP1:90,1] + -33.071;
   1:  PR[GP1:91,2] = PR[GP1:90,2] + -36.283;
   1:L PR[91] 10mm/sec CNT100;
   1:  PR[GP1:91,1] = PR[GP1:90,1] + -32.743;
   1:  PR[GP1:91,2] = PR[GP1:90,2] + -36.611;
   1:L PR[91] 10mm/sec CNT100;
   1:  PR[GP1:91,1] = PR[GP1:90,1] + -23.136;
   1:  PR[GP1:91,2] = PR[GP1:90,2] + -43.413;
   1:L PR[91] 10mm/sec CNT100;
   1:  PR[GP1:91,1] = PR[GP1:90,1] + -22.721;
   1:  PR[GP1:91,2] = PR[GP1:90,2] + -43.624;
   1:L PR[91] 10mm/sec CNT100;
   1:  PR[GP1:91,1] = PR[GP1:90,1] + -11.755;
   1:  PR[GP1:91,2] = PR[GP1:90,2] + -47.874;
   1:L PR[91] 10mm/sec CNT100;
   1:  PR[GP1:91,1] = PR[GP1:90,1] + -0.041;
   1:  PR[GP1:91,2] = PR[GP1:90,2] + -49.326;
   1:L PR[91] 10mm/sec CNT100;
   1:  PR[GP1:91,1] = PR[GP1:90,1] + 0.419;
   1:  PR[GP1:91,2] = PR[GP1:90,2] + -49.399;
   1:L PR[91] 10mm/sec CNT100;
   1:  PR[GP1:91,1] = PR[GP1:90,1] + 12.104;
   1:  PR[GP1:91,2] = PR[GP1:90,2] + -47.951;
   1:L PR[91] 10mm/sec CNT100;
   1:  PR[GP1:91,1] = PR[GP1:90,1] + 12.564;
   1:  PR[GP1:91,2] = PR[GP1:90,2] + -47.879;
   1:L PR[91] 10mm/sec CNT100;
   1:  PR[GP1:91,1] = PR[GP1:90,1] + 23.542;
   1:  PR[GP1:91,2] = PR[GP1:90,2] + -43.625;
   1:L PR[91] 10mm/sec CNT100;
   1:  PR[GP1:91,1] = PR[GP1:90,1] + 23.957;
   1:  PR[GP1:91,2] = PR[GP1:90,2] + -43.413;
   1:L PR[91] 10mm/sec CNT100;
   1:  PR[GP1:91,1] = PR[GP1:90,1] + 33.566;
   1:  PR[GP1:91,2] = PR[GP1:90,2] + -36.609;
   1:L PR[91] 10mm/sec CNT100;
   1:  PR[GP1:91,1] = PR[GP1:90,1] + 33.891;
   1:  PR[GP1:91,2] = PR[GP1:90,2] + -36.284;
   1:L PR[91] 10mm/sec CNT100;
   1:  PR[GP1:91,1] = PR[GP1:90,1] + 42.349;
   1:  PR[GP1:91,2] = PR[GP1:90,2] + -26.096;
   1:L PR[91] 10mm/sec CNT100;
   1:  PR[GP1:91,1] = PR[GP1:90,1] + 42.556;
   1:  PR[GP1:91,2] = PR[GP1:90,2] + -25.689;
   1:L PR[91] 10mm/sec CNT100;
   1:  PR[GP1:91,1] = PR[GP1:90,1] + 47.901;
   1:  PR[GP1:91,2] = PR[GP1:90,2] + -13.581;
   1:L PR[91] 10mm/sec CNT100;
   1:  PR[GP1:91,1] = PR[GP1:90,1] + 49.804;
   1:  PR[GP1:91,2] = PR[GP1:90,2] + -0.004;
   1:L PR[91] 10mm/sec CNT100;
   1:  PR[GP1:91,1] = PR[GP1:90,1] + 47.901;
   1:  PR[GP1:91,2] = PR[GP1:90,2] + 13.572;
   1:L PR[91] 10mm/sec CNT100;
   1:  PR[GP1:91,1] = PR[GP1:90,1] + 42.556;
   1:  PR[GP1:91,2] = PR[GP1:90,2] + 25.680;
   1:L PR[91] 10mm/sec CNT100;
   1:  PR[GP1:91,1] = PR[GP1:90,1] + 42.349;
   1:  PR[GP1:91,2] = PR[GP1:90,2] + 26.087;
   1:L PR[91] 10mm/sec CNT100;
   1:  PR[GP1:91,1] = PR[GP1:90,1] + 33.891;
   1:  PR[GP1:91,2] = PR[GP1:90,2] + 36.275;
   1:L PR[91] 10mm/sec CNT100;
   1:  PR[GP1:91,1] = PR[GP1:90,1] + 33.566;
   1:  PR[GP1:91,2] = PR[GP1:90,2] + 36.600;
   1:L PR[91] 10mm/sec CNT100;
   1:  PR[GP1:91,1] = PR[GP1:90,1] + 23.957;
   1:  PR[GP1:91,2] = PR[GP1:90,2] + 43.404;
   1:L PR[91] 10mm/sec CNT100;
   1:  PR[GP1:91,1] = PR[GP1:90,1] + 23.542;
   1:  PR[GP1:91,2] = PR[GP1:90,2] + 43.616;
   1:L PR[91] 10mm/sec CNT100;
   1:  PR[GP1:91,1] = PR[GP1:90,1] + 12.564;
   1:  PR[GP1:91,2] = PR[GP1:90,2] + 47.870;
   1:L PR[91] 10mm/sec CNT100;
   1:  PR[GP1:91,1] = PR[GP1:90,1] + 12.104;
   1:  PR[GP1:91,2] = PR[GP1:90,2] + 47.943;
   1:L PR[91] 10mm/sec CNT100;
   1:  PR[GP1:91,1] = PR[GP1:90,1] + 0.408;
   1:  PR[GP1:91,2] = PR[GP1:90,2] + 49.391;
   1:L PR[91] 10mm/sec CNT100;
   1:  PR[GP1:91,1] = PR[GP1:90,1] + -9.663;
   1:  PR[GP1:91,2] = PR[GP1:90,2] + 48.143;
   1:  PR[GP1:91,3] = PR[GP1:90,3] + 130.340;
   1:L PR[91] 10mm/sec CNT100;
   1:  PR[GP1:91,1] = PR[GP1:90,1] + -12.178;
   1:  PR[GP1:91,2] = PR[GP1:90,2] + 47.745;
   1:L PR[91] 10mm/sec CNT100;
   1:  PR[GP1:91,1] = PR[GP1:90,1] + -21.630;
   1:  PR[GP1:91,2] = PR[GP1:90,2] + 44.082;
   1:L PR[91] 10mm/sec CNT100;
   1:  PR[GP1:91,1] = PR[GP1:90,1] + -23.898;
   1:  PR[GP1:91,2] = PR[GP1:90,2] + 42.926;
   1:L PR[91] 10mm/sec CNT100;
   1:  PR[GP1:91,1] = PR[GP1:90,1] + -32.171;
   1:  PR[GP1:91,2] = PR[GP1:90,2] + 37.068;
   1:L PR[91] 10mm/sec CNT100;
   1:  PR[GP1:91,1] = PR[GP1:90,1] + -33.970;
   1:  PR[GP1:91,2] = PR[GP1:90,2] + 35.270;
   1:L PR[91] 10mm/sec CNT100;
   1:  PR[GP1:91,1] = PR[GP1:90,1] + -41.253;
   1:  PR[GP1:91,2] = PR[GP1:90,2] + 26.496;
   1:L PR[91] 10mm/sec CNT100;
   1:  PR[GP1:91,1] = PR[GP1:90,1] + -42.405;
   1:  PR[GP1:91,2] = PR[GP1:90,2] + 24.236;
   1:L PR[91] 10mm/sec CNT100;
   1:  PR[GP1:91,1] = PR[GP1:90,1] + -47.008;
   1:  PR[GP1:91,2] = PR[GP1:90,2] + 13.808;
   1:L PR[91] 10mm/sec CNT100;
   1:  PR[GP1:91,1] = PR[GP1:90,1] + -48.586;
   1:  PR[GP1:91,2] = PR[GP1:90,2] + 2.495;
   1:L PR[91] 10mm/sec CNT100;
   1:  PR[GP1:91,1] = PR[GP1:90,1] + -48.983;
   1:  PR[GP1:91,2] = PR[GP1:90,2] + -0.010;
   1:L PR[91] 10mm/sec CNT100;
   1:  PR[GP1:91,1] = PR[GP1:90,1] + -47.407;
   1:  PR[GP1:91,2] = PR[GP1:90,2] + -11.306;
   1:L PR[91] 10mm/sec CNT100;
   1:  PR[GP1:91,1] = PR[GP1:90,1] + -47.011;
   1:  PR[GP1:91,2] = PR[GP1:90,2] + -13.811;
   1:L PR[91] 10mm/sec CNT100;
   1:  PR[GP1:91,1] = PR[GP1:90,1] + -42.405;
   1:  PR[GP1:91,2] = PR[GP1:90,2] + -24.245;
   1:L PR[91] 10mm/sec CNT100;
   1:  PR[GP1:91,1] = PR[GP1:90,1] + -41.253;
   1:  PR[GP1:91,2] = PR[GP1:90,2] + -26.505;
   1:L PR[91] 10mm/sec CNT100;
   1:  PR[GP1:91,1] = PR[GP1:90,1] + -33.969;
   1:  PR[GP1:91,2] = PR[GP1:90,2] + -35.278;
   1:L PR[91] 10mm/sec CNT100;
   1:  PR[GP1:91,1] = PR[GP1:90,1] + -32.171;
   1:  PR[GP1:91,2] = PR[GP1:90,2] + -37.077;
   1:L PR[91] 10mm/sec CNT100;
   1:  PR[GP1:91,1] = PR[GP1:90,1] + -23.898;
   1:  PR[GP1:91,2] = PR[GP1:90,2] + -42.935;
   1:L PR[91] 10mm/sec CNT100;
   1:  PR[GP1:91,1] = PR[GP1:90,1] + -21.630;
   1:  PR[GP1:91,2] = PR[GP1:90,2] + -44.091;
   1:L PR[91] 10mm/sec CNT100;
   1:  PR[GP1:91,1] = PR[GP1:90,1] + -12.187;
   1:  PR[GP1:91,2] = PR[GP1:90,2] + -47.750;
   1:L PR[91] 10mm/sec CNT100;
   1:  PR[GP1:91,1] = PR[GP1:90,1] + -2.096;
   1:  PR[GP1:91,2] = PR[GP1:90,2] + -49.000;
   1:L PR[91] 10mm/sec CNT100;
   1:  PR[GP1:91,1] = PR[GP1:90,1] + 0.419;
   1:  PR[GP1:91,2] = PR[GP1:90,2] + -49.399;
   1:L PR[91] 10mm/sec CNT100;
   1:  PR[GP1:91,1] = PR[GP1:90,1] + 10.482;
   1:  PR[GP1:91,2] = PR[GP1:90,2] + -48.152;
   1:L PR[91] 10mm/sec CNT100;
   1:  PR[GP1:91,1] = PR[GP1:90,1] + 12.997;
   1:  PR[GP1:91,2] = PR[GP1:90,2] + -47.754;
   1:L PR[91] 10mm/sec CNT100;
   1:  PR[GP1:91,1] = PR[GP1:90,1] + 22.450;
   1:  PR[GP1:91,2] = PR[GP1:90,2] + -44.091;
   1:L PR[91] 10mm/sec CNT100;
   1:  PR[GP1:91,1] = PR[GP1:90,1] + 24.719;
   1:  PR[GP1:91,2] = PR[GP1:90,2] + -42.935;
   1:L PR[91] 10mm/sec CNT100;
   1:  PR[GP1:91,1] = PR[GP1:90,1] + 32.993;
   1:  PR[GP1:91,2] = PR[GP1:90,2] + -37.075;
   1:L PR[91] 10mm/sec CNT100;
   1:  PR[GP1:91,1] = PR[GP1:90,1] + 34.790;
   1:  PR[GP1:91,2] = PR[GP1:90,2] + -35.279;
   1:L PR[91] 10mm/sec CNT100;
   1:  PR[GP1:91,1] = PR[GP1:90,1] + 42.074;
   1:  PR[GP1:91,2] = PR[GP1:90,2] + -26.504;
   1:L PR[91] 10mm/sec CNT100;
   1:  PR[GP1:91,1] = PR[GP1:90,1] + 43.226;
   1:  PR[GP1:91,2] = PR[GP1:90,2] + -24.244;
   1:L PR[91] 10mm/sec CNT100;
   1:  PR[GP1:91,1] = PR[GP1:90,1] + 47.829;
   1:  PR[GP1:91,2] = PR[GP1:90,2] + -13.816;
   1:L PR[91] 10mm/sec CNT100;
   1:  PR[GP1:91,1] = PR[GP1:90,1] + 49.407;
   1:  PR[GP1:91,2] = PR[GP1:90,2] + -2.504;
   1:L PR[91] 10mm/sec CNT100;
   1:  PR[GP1:91,1] = PR[GP1:90,1] + 49.804;
   1:  PR[GP1:91,2] = PR[GP1:90,2] + 0.001;
   1:L PR[91] 10mm/sec CNT100;
   1:  PR[GP1:91,1] = PR[GP1:90,1] + 48.228;
   1:  PR[GP1:91,2] = PR[GP1:90,2] + 11.297;
   1:L PR[91] 10mm/sec CNT100;
   1:  PR[GP1:91,1] = PR[GP1:90,1] + 47.831;
   1:  PR[GP1:91,2] = PR[GP1:90,2] + 13.802;
   1:L PR[91] 10mm/sec CNT100;
   1:  PR[GP1:91,1] = PR[GP1:90,1] + 43.226;
   1:  PR[GP1:91,2] = PR[GP1:90,2] + 24.235;
   1:L PR[91] 10mm/sec CNT100;
   1:  PR[GP1:91,1] = PR[GP1:90,1] + 42.074;
   1:  PR[GP1:91,2] = PR[GP1:90,2] + 26.495;
   1:L PR[91] 10mm/sec CNT100;
   1:  PR[GP1:91,1] = PR[GP1:90,1] + 34.790;
   1:  PR[GP1:91,2] = PR[GP1:90,2] + 35.270;
   1:L PR[91] 10mm/sec CNT100;
   1:  PR[GP1:91,1] = PR[GP1:90,1] + 32.993;
   1:  PR[GP1:91,2] = PR[GP1:90,2] + 37.067;
   1:L PR[91] 10mm/sec CNT100;
   1:  PR[GP1:91,1] = PR[GP1:90,1] + 24.719;
   1:  PR[GP1:91,2] = PR[GP1:90,2] + 42.926;
   1:L PR[91] 10mm/sec CNT100;
   1:  PR[GP1:91,1] = PR[GP1:90,1] + 22.450;
   1:  PR[GP1:91,2] = PR[GP1:90,2] + 44.082;
   1:L PR[91] 10mm/sec CNT100;
   1:  PR[GP1:91,1] = PR[GP1:90,1] + 12.997;
   1:  PR[GP1:91,2] = PR[GP1:90,2] + 47.745;
   1:L PR[91] 10mm/sec CNT100;
   1:  PR[GP1:91,1] = PR[GP1:90,1] + 10.482;
   1:  PR[GP1:91,2] = PR[GP1:90,2] + 48.144;
   1:L PR[91] 10mm/sec CNT100;
   1:  PR[GP1:91,1] = PR[GP1:90,1] + 0.409;
   1:  PR[GP1:91,2] = PR[GP1:90,2] + 49.391;
   1:L PR[91] 10mm/sec CNT100;
   1:  PR[GP1:91,1] = PR[GP1:90,1] + -8.040;
   1:  PR[GP1:91,2] = PR[GP1:90,2] + 48.344;
   1:  PR[GP1:91,3] = PR[GP1:90,3] + 131.670;
   1:L PR[91] 10mm/sec CNT100;
   1:  PR[GP1:91,1] = PR[GP1:90,1] + -12.610;
   1:  PR[GP1:91,2] = PR[GP1:90,2] + 47.620;
   1:L PR[91] 10mm/sec CNT100;
   1:  PR[GP1:91,1] = PR[GP1:90,1] + -20.538;
   1:  PR[GP1:91,2] = PR[GP1:90,2] + 44.548;
   1:L PR[91] 10mm/sec CNT100;
   1:  PR[GP1:91,1] = PR[GP1:90,1] + -24.660;
   1:  PR[GP1:91,2] = PR[GP1:90,2] + 42.447;
   1:L PR[91] 10mm/sec CNT100;
   1:  PR[GP1:91,1] = PR[GP1:90,1] + -31.599;
   1:  PR[GP1:91,2] = PR[GP1:90,2] + 37.534;
   1:L PR[91] 10mm/sec CNT100;
   1:  PR[GP1:91,1] = PR[GP1:90,1] + -34.868;
   1:  PR[GP1:91,2] = PR[GP1:90,2] + 34.265;
   1:L PR[91] 10mm/sec CNT100;
   1:  PR[GP1:91,1] = PR[GP1:90,1] + -40.979;
   1:  PR[GP1:91,2] = PR[GP1:90,2] + 26.905;
   1:L PR[91] 10mm/sec CNT100;
   1:  PR[GP1:91,1] = PR[GP1:90,1] + -43.075;
   1:  PR[GP1:91,2] = PR[GP1:90,2] + 22.790;
   1:L PR[91] 10mm/sec CNT100;
   1:  PR[GP1:91,1] = PR[GP1:90,1] + -46.937;
   1:  PR[GP1:91,2] = PR[GP1:90,2] + 14.043;
   1:L PR[91] 10mm/sec CNT100;
   1:  PR[GP1:91,1] = PR[GP1:90,1] + -48.261;
   1:  PR[GP1:91,2] = PR[GP1:90,2] + 4.550;
   1:L PR[91] 10mm/sec CNT100;
   1:  PR[GP1:91,1] = PR[GP1:90,1] + -48.983;
   1:  PR[GP1:91,2] = PR[GP1:90,2] + -0.010;
   1:L PR[91] 10mm/sec CNT100;
   1:  PR[GP1:91,1] = PR[GP1:90,1] + -47.661;
   1:  PR[GP1:91,2] = PR[GP1:90,2] + -9.487;
   1:L PR[91] 10mm/sec CNT100;
   1:  PR[GP1:91,1] = PR[GP1:90,1] + -46.939;
   1:  PR[GP1:91,2] = PR[GP1:90,2] + -14.047;
   1:L PR[91] 10mm/sec CNT100;
   1:  PR[GP1:91,1] = PR[GP1:90,1] + -43.075;
   1:  PR[GP1:91,2] = PR[GP1:90,2] + -22.799;
   1:L PR[91] 10mm/sec CNT100;
   1:  PR[GP1:91,1] = PR[GP1:90,1] + -40.979;
   1:  PR[GP1:91,2] = PR[GP1:90,2] + -26.913;
   1:L PR[91] 10mm/sec CNT100;
   1:  PR[GP1:91,1] = PR[GP1:90,1] + -34.868;
   1:  PR[GP1:91,2] = PR[GP1:90,2] + -34.274;
   1:L PR[91] 10mm/sec CNT100;
   1:  PR[GP1:91,1] = PR[GP1:90,1] + -31.599;
   1:  PR[GP1:91,2] = PR[GP1:90,2] + -37.543;
   1:L PR[91] 10mm/sec CNT100;
   1:  PR[GP1:91,1] = PR[GP1:90,1] + -24.660;
   1:  PR[GP1:91,2] = PR[GP1:90,2] + -42.456;
   1:L PR[91] 10mm/sec CNT100;
   1:  PR[GP1:91,1] = PR[GP1:90,1] + -20.538;
   1:  PR[GP1:91,2] = PR[GP1:90,2] + -44.557;
   1:L PR[91] 10mm/sec CNT100;
   1:  PR[GP1:91,1] = PR[GP1:90,1] + -12.620;
   1:  PR[GP1:91,2] = PR[GP1:90,2] + -47.625;
   1:L PR[91] 10mm/sec CNT100;
   1:  PR[GP1:91,1] = PR[GP1:90,1] + -4.150;
   1:  PR[GP1:91,2] = PR[GP1:90,2] + -48.675;
   1:L PR[91] 10mm/sec CNT100;
   1:  PR[GP1:91,1] = PR[GP1:90,1] + 0.419;
   1:  PR[GP1:91,2] = PR[GP1:90,2] + -49.399;
   1:L PR[91] 10mm/sec CNT100;
   1:  PR[GP1:91,1] = PR[GP1:90,1] + 8.859;
   1:  PR[GP1:91,2] = PR[GP1:90,2] + -48.353;
   1:L PR[91] 10mm/sec CNT100;
   1:  PR[GP1:91,1] = PR[GP1:90,1] + 13.429;
   1:  PR[GP1:91,2] = PR[GP1:90,2] + -47.630;
   1:L PR[91] 10mm/sec CNT100;
   1:  PR[GP1:91,1] = PR[GP1:90,1] + 21.358;
   1:  PR[GP1:91,2] = PR[GP1:90,2] + -44.557;
   1:L PR[91] 10mm/sec CNT100;
   1:  PR[GP1:91,1] = PR[GP1:90,1] + 25.481;
   1:  PR[GP1:91,2] = PR[GP1:90,2] + -42.456;
   1:L PR[91] 10mm/sec CNT100;
   1:  PR[GP1:91,1] = PR[GP1:90,1] + 32.421;
   1:  PR[GP1:91,2] = PR[GP1:90,2] + -37.542;
   1:L PR[91] 10mm/sec CNT100;
   1:  PR[GP1:91,1] = PR[GP1:90,1] + 35.689;
   1:  PR[GP1:91,2] = PR[GP1:90,2] + -34.274;
   1:L PR[91] 10mm/sec CNT100;
   1:  PR[GP1:91,1] = PR[GP1:90,1] + 41.800;
   1:  PR[GP1:91,2] = PR[GP1:90,2] + -26.913;
   1:L PR[91] 10mm/sec CNT100;
   1:  PR[GP1:91,1] = PR[GP1:90,1] + 43.896;
   1:  PR[GP1:91,2] = PR[GP1:90,2] + -22.799;
   1:L PR[91] 10mm/sec CNT100;
   1:  PR[GP1:91,1] = PR[GP1:90,1] + 47.757;
   1:  PR[GP1:91,2] = PR[GP1:90,2] + -14.052;
   1:L PR[91] 10mm/sec CNT100;
   1:  PR[GP1:91,1] = PR[GP1:90,1] + 49.081;
   1:  PR[GP1:91,2] = PR[GP1:90,2] + -4.559;
   1:L PR[91] 10mm/sec CNT100;
   1:  PR[GP1:91,1] = PR[GP1:90,1] + 49.804;
   1:  PR[GP1:91,2] = PR[GP1:90,2] + 0.001;
   1:L PR[91] 10mm/sec CNT100;
   1:  PR[GP1:91,1] = PR[GP1:90,1] + 48.482;
   1:  PR[GP1:91,2] = PR[GP1:90,2] + 9.478;
   1:L PR[91] 10mm/sec CNT100;
   1:  PR[GP1:91,1] = PR[GP1:90,1] + 47.760;
   1:  PR[GP1:91,2] = PR[GP1:90,2] + 14.038;
   1:L PR[91] 10mm/sec CNT100;
   1:  PR[GP1:91,1] = PR[GP1:90,1] + 43.896;
   1:  PR[GP1:91,2] = PR[GP1:90,2] + 22.790;
   1:L PR[91] 10mm/sec CNT100;
   1:  PR[GP1:91,1] = PR[GP1:90,1] + 41.800;
   1:  PR[GP1:91,2] = PR[GP1:90,2] + 26.904;
   1:L PR[91] 10mm/sec CNT100;
   1:  PR[GP1:91,1] = PR[GP1:90,1] + 35.689;
   1:  PR[GP1:91,2] = PR[GP1:90,2] + 34.265;
   1:L PR[91] 10mm/sec CNT100;
   1:  PR[GP1:91,1] = PR[GP1:90,1] + 32.421;
   1:  PR[GP1:91,2] = PR[GP1:90,2] + 37.533;
   1:L PR[91] 10mm/sec CNT100;
   1:  PR[GP1:91,1] = PR[GP1:90,1] + 25.481;
   1:  PR[GP1:91,2] = PR[GP1:90,2] + 42.448;
   1:L PR[91] 10mm/sec CNT100;
   1:  PR[GP1:91,1] = PR[GP1:90,1] + 21.358;
   1:  PR[GP1:91,2] = PR[GP1:90,2] + 44.548;
   1:L PR[91] 10mm/sec CNT100;
   1:  PR[GP1:91,1] = PR[GP1:90,1] + 13.429;
   1:  PR[GP1:91,2] = PR[GP1:90,2] + 47.621;
   1:L PR[91] 10mm/sec CNT100;
   1:  PR[GP1:91,1] = PR[GP1:90,1] + 8.859;
   1:  PR[GP1:91,2] = PR[GP1:90,2] + 48.344;
   1:L PR[91] 10mm/sec CNT100;
   1:  PR[GP1:91,1] = PR[GP1:90,1] + 0.409;
   1:  PR[GP1:91,2] = PR[GP1:90,2] + 49.391;
   1:L PR[91] 10mm/sec CNT100;
   1:  PR[GP1:91,1] = PR[GP1:90,1] + -6.418;
   1:  PR[GP1:91,2] = PR[GP1:90,2] + 48.545;
   1:  PR[GP1:91,3] = PR[GP1:90,3] + 133.000;
   1:L PR[91] 10mm/sec CNT100;
   1:  PR[GP1:91,1] = PR[GP1:90,1] + -13.042;
   1:  PR[GP1:91,2] = PR[GP1:90,2] + 47.496;
   1:L PR[91] 10mm/sec CNT100;
   1:  PR[GP1:91,1] = PR[GP1:90,1] + -19.446;
   1:  PR[GP1:91,2] = PR[GP1:90,2] + 45.014;
   1:L PR[91] 10mm/sec CNT100;
   1:  PR[GP1:91,1] = PR[GP1:90,1] + -25.422;
   1:  PR[GP1:91,2] = PR[GP1:90,2] + 41.969;
   1:L PR[91] 10mm/sec CNT100;
   1:  PR[GP1:91,1] = PR[GP1:90,1] + -31.027;
   1:  PR[GP1:91,2] = PR[GP1:90,2] + 38.000;
   1:L PR[91] 10mm/sec CNT100;
   1:  PR[GP1:91,1] = PR[GP1:90,1] + -35.767;
   1:  PR[GP1:91,2] = PR[GP1:90,2] + 33.260;
   1:L PR[91] 10mm/sec CNT100;
   1:  PR[GP1:91,1] = PR[GP1:90,1] + -40.705;
   1:  PR[GP1:91,2] = PR[GP1:90,2] + 27.313;
   1:L PR[91] 10mm/sec CNT100;
   1:  PR[GP1:91,1] = PR[GP1:90,1] + -43.745;
   1:  PR[GP1:91,2] = PR[GP1:90,2] + 21.345;
   1:L PR[91] 10mm/sec CNT100;
   1:  PR[GP1:91,1] = PR[GP1:90,1] + -46.865;
   1:  PR[GP1:91,2] = PR[GP1:90,2] + 14.278;
   1:L PR[91] 10mm/sec CNT100;
   1:  PR[GP1:91,1] = PR[GP1:90,1] + -47.935;
   1:  PR[GP1:91,2] = PR[GP1:90,2] + 6.605;
   1:L PR[91] 10mm/sec CNT100;
   1:  PR[GP1:91,1] = PR[GP1:90,1] + -48.983;
   1:  PR[GP1:91,2] = PR[GP1:90,2] + -0.010;
   1:L PR[91] 10mm/sec CNT100;
   1:  PR[GP1:91,1] = PR[GP1:90,1] + -47.915;
   1:  PR[GP1:91,2] = PR[GP1:90,2] + -7.667;
   1:L PR[91] 10mm/sec CNT100;
   1:  PR[GP1:91,1] = PR[GP1:90,1] + -46.867;
   1:  PR[GP1:91,2] = PR[GP1:90,2] + -14.282;
   1:L PR[91] 10mm/sec CNT100;
   1:  PR[GP1:91,1] = PR[GP1:90,1] + -43.745;
   1:  PR[GP1:91,2] = PR[GP1:90,2] + -21.354;
   1:L PR[91] 10mm/sec CNT100;
   1:  PR[GP1:91,1] = PR[GP1:90,1] + -40.705;
   1:  PR[GP1:91,2] = PR[GP1:90,2] + -27.322;
   1:L PR[91] 10mm/sec CNT100;
   1:  PR[GP1:91,1] = PR[GP1:90,1] + -35.767;
   1:  PR[GP1:91,2] = PR[GP1:90,2] + -33.269;
   1:L PR[91] 10mm/sec CNT100;
   1:  PR[GP1:91,1] = PR[GP1:90,1] + -31.027;
   1:  PR[GP1:91,2] = PR[GP1:90,2] + -38.009;
   1:L PR[91] 10mm/sec CNT100;
   1:  PR[GP1:91,1] = PR[GP1:90,1] + -25.422;
   1:  PR[GP1:91,2] = PR[GP1:90,2] + -41.978;
   1:L PR[91] 10mm/sec CNT100;
   1:  PR[GP1:91,1] = PR[GP1:90,1] + -19.446;
   1:  PR[GP1:91,2] = PR[GP1:90,2] + -45.023;
   1:L PR[91] 10mm/sec CNT100;
   1:  PR[GP1:91,1] = PR[GP1:90,1] + -13.052;
   1:  PR[GP1:91,2] = PR[GP1:90,2] + -47.501;
   1:L PR[91] 10mm/sec CNT100;
   1:  PR[GP1:91,1] = PR[GP1:90,1] + -6.205;
   1:  PR[GP1:91,2] = PR[GP1:90,2] + -48.349;
   1:L PR[91] 10mm/sec CNT100;
   1:  PR[GP1:91,1] = PR[GP1:90,1] + 0.419;
   1:  PR[GP1:91,2] = PR[GP1:90,2] + -49.399;
   1:L PR[91] 10mm/sec CNT100;
   1:  PR[GP1:91,1] = PR[GP1:90,1] + 7.237;
   1:  PR[GP1:91,2] = PR[GP1:90,2] + -48.554;
   1:L PR[91] 10mm/sec CNT100;
   1:  PR[GP1:91,1] = PR[GP1:90,1] + 13.862;
   1:  PR[GP1:91,2] = PR[GP1:90,2] + -47.505;
   1:L PR[91] 10mm/sec CNT100;
   1:  PR[GP1:91,1] = PR[GP1:90,1] + 20.266;
   1:  PR[GP1:91,2] = PR[GP1:90,2] + -45.023;
   1:L PR[91] 10mm/sec CNT100;
   1:  PR[GP1:91,1] = PR[GP1:90,1] + 26.243;
   1:  PR[GP1:91,2] = PR[GP1:90,2] + -41.978;
   1:L PR[91] 10mm/sec CNT100;
   1:  PR[GP1:91,1] = PR[GP1:90,1] + 31.849;
   1:  PR[GP1:91,2] = PR[GP1:90,2] + -38.008;
   1:L PR[91] 10mm/sec CNT100;
   1:  PR[GP1:91,1] = PR[GP1:90,1] + 36.588;
   1:  PR[GP1:91,2] = PR[GP1:90,2] + -33.269;
   1:L PR[91] 10mm/sec CNT100;
   1:  PR[GP1:91,1] = PR[GP1:90,1] + 41.525;
   1:  PR[GP1:91,2] = PR[GP1:90,2] + -27.321;
   1:L PR[91] 10mm/sec CNT100;
   1:  PR[GP1:91,1] = PR[GP1:90,1] + 44.566;
   1:  PR[GP1:91,2] = PR[GP1:90,2] + -21.354;
   1:L PR[91] 10mm/sec CNT100;
   1:  PR[GP1:91,1] = PR[GP1:90,1] + 47.686;
   1:  PR[GP1:91,2] = PR[GP1:90,2] + -14.287;
   1:L PR[91] 10mm/sec CNT100;
   1:  PR[GP1:91,1] = PR[GP1:90,1] + 48.756;
   1:  PR[GP1:91,2] = PR[GP1:90,2] + -6.614;
   1:L PR[91] 10mm/sec CNT100;
   1:  PR[GP1:91,1] = PR[GP1:90,1] + 49.804;
   1:  PR[GP1:91,2] = PR[GP1:90,2] + 0.001;
   1:L PR[91] 10mm/sec CNT100;
   1:  PR[GP1:91,1] = PR[GP1:90,1] + 48.736;
   1:  PR[GP1:91,2] = PR[GP1:90,2] + 7.658;
   1:L PR[91] 10mm/sec CNT100;
   1:  PR[GP1:91,1] = PR[GP1:90,1] + 47.688;
   1:  PR[GP1:91,2] = PR[GP1:90,2] + 14.273;
   1:L PR[91] 10mm/sec CNT100;
   1:  PR[GP1:91,1] = PR[GP1:90,1] + 44.566;
   1:  PR[GP1:91,2] = PR[GP1:90,2] + 21.345;
   1:L PR[91] 10mm/sec CNT100;
   1:  PR[GP1:91,1] = PR[GP1:90,1] + 41.525;
   1:  PR[GP1:91,2] = PR[GP1:90,2] + 27.312;
   1:L PR[91] 10mm/sec CNT100;
   1:  PR[GP1:91,1] = PR[GP1:90,1] + 36.588;
   1:  PR[GP1:91,2] = PR[GP1:90,2] + 33.260;
   1:L PR[91] 10mm/sec CNT100;
   1:  PR[GP1:91,1] = PR[GP1:90,1] + 31.849;
   1:  PR[GP1:91,2] = PR[GP1:90,2] + 37.999;
   1:L PR[91] 10mm/sec CNT100;
   1:  PR[GP1:91,1] = PR[GP1:90,1] + 26.243;
   1:  PR[GP1:91,2] = PR[GP1:90,2] + 41.969;
   1:L PR[91] 10mm/sec CNT100;
   1:  PR[GP1:91,1] = PR[GP1:90,1] + 20.266;
   1:  PR[GP1:91,2] = PR[GP1:90,2] + 45.014;
   1:L PR[91] 10mm/sec CNT100;
   1:  PR[GP1:91,1] = PR[GP1:90,1] + 13.862;
   1:  PR[GP1:91,2] = PR[GP1:90,2] + 47.496;
   1:L PR[91] 10mm/sec CNT100;
   1:  PR[GP1:91,1] = PR[GP1:90,1] + 7.237;
   1:  PR[GP1:91,2] = PR[GP1:90,2] + 48.545;
   1:L PR[91] 10mm/sec CNT100;
   1:  PR[GP1:91,1] = PR[GP1:90,1] + 0.409;
   1:  PR[GP1:91,2] = PR[GP1:90,2] + 49.391;
   1:L PR[91] 10mm/sec CNT100;
   1:  PR[GP1:91,1] = PR[GP1:90,1] + -4.795;
   1:  PR[GP1:91,2] = PR[GP1:90,2] + 48.746;
   1:  PR[GP1:91,3] = PR[GP1:90,3] + 134.330;
   1:L PR[91] 10mm/sec CNT100;
   1:  PR[GP1:91,1] = PR[GP1:90,1] + -13.474;
   1:  PR[GP1:91,2] = PR[GP1:90,2] + 47.371;
   1:L PR[91] 10mm/sec CNT100;
   1:  PR[GP1:91,1] = PR[GP1:90,1] + -18.354;
   1:  PR[GP1:91,2] = PR[GP1:90,2] + 45.480;
   1:L PR[91] 10mm/sec CNT100;
   1:  PR[GP1:91,1] = PR[GP1:90,1] + -26.184;
   1:  PR[GP1:91,2] = PR[GP1:90,2] + 41.491;
   1:L PR[91] 10mm/sec CNT100;
   1:  PR[GP1:91,1] = PR[GP1:90,1] + -30.455;
   1:  PR[GP1:91,2] = PR[GP1:90,2] + 38.467;
   1:L PR[91] 10mm/sec CNT100;
   1:  PR[GP1:91,1] = PR[GP1:90,1] + -36.666;
   1:  PR[GP1:91,2] = PR[GP1:90,2] + 32.255;
   1:L PR[91] 10mm/sec CNT100;
   1:  PR[GP1:91,1] = PR[GP1:90,1] + -40.430;
   1:  PR[GP1:91,2] = PR[GP1:90,2] + 27.721;
   1:L PR[91] 10mm/sec CNT100;
   1:  PR[GP1:91,1] = PR[GP1:90,1] + -44.416;
   1:  PR[GP1:91,2] = PR[GP1:90,2] + 19.900;
   1:L PR[91] 10mm/sec CNT100;
   1:  PR[GP1:91,1] = PR[GP1:90,1] + -46.793;
   1:  PR[GP1:91,2] = PR[GP1:90,2] + 14.514;
   1:L PR[91] 10mm/sec CNT100;
   1:  PR[GP1:91,1] = PR[GP1:90,1] + -47.610;
   1:  PR[GP1:91,2] = PR[GP1:90,2] + 8.660;
   1:L PR[91] 10mm/sec CNT100;
   1:  PR[GP1:91,1] = PR[GP1:90,1] + -48.983;
   1:  PR[GP1:91,2] = PR[GP1:90,2] + -0.010;
   1:L PR[91] 10mm/sec CNT100;
   1:  PR[GP1:91,1] = PR[GP1:90,1] + -48.169;
   1:  PR[GP1:91,2] = PR[GP1:90,2] + -5.847;
   1:L PR[91] 10mm/sec CNT100;
   1:  PR[GP1:91,1] = PR[GP1:90,1] + -46.796;
   1:  PR[GP1:91,2] = PR[GP1:90,2] + -14.517;
   1:L PR[91] 10mm/sec CNT100;
   1:  PR[GP1:91,1] = PR[GP1:90,1] + -44.416;
   1:  PR[GP1:91,2] = PR[GP1:90,2] + -19.909;
   1:L PR[91] 10mm/sec CNT100;
   1:  PR[GP1:91,1] = PR[GP1:90,1] + -40.430;
   1:  PR[GP1:91,2] = PR[GP1:90,2] + -27.730;
   1:L PR[91] 10mm/sec CNT100;
   1:  PR[GP1:91,1] = PR[GP1:90,1] + -36.666;
   1:  PR[GP1:91,2] = PR[GP1:90,2] + -32.264;
   1:L PR[91] 10mm/sec CNT100;
   1:  PR[GP1:91,1] = PR[GP1:90,1] + -30.455;
   1:  PR[GP1:91,2] = PR[GP1:90,2] + -38.475;
   1:L PR[91] 10mm/sec CNT100;
   1:  PR[GP1:91,1] = PR[GP1:90,1] + -26.184;
   1:  PR[GP1:91,2] = PR[GP1:90,2] + -41.500;
   1:L PR[91] 10mm/sec CNT100;
   1:  PR[GP1:91,1] = PR[GP1:90,1] + -18.354;
   1:  PR[GP1:91,2] = PR[GP1:90,2] + -45.489;
   1:L PR[91] 10mm/sec CNT100;
   1:  PR[GP1:91,1] = PR[GP1:90,1] + -13.484;
   1:  PR[GP1:91,2] = PR[GP1:90,2] + -47.377;
   1:L PR[91] 10mm/sec CNT100;
   1:  PR[GP1:91,1] = PR[GP1:90,1] + -8.260;
   1:  PR[GP1:91,2] = PR[GP1:90,2] + -48.024;
   1:L PR[91] 10mm/sec CNT100;
   1:  PR[GP1:91,1] = PR[GP1:90,1] + 0.420;
   1:  PR[GP1:91,2] = PR[GP1:90,2] + -49.399;
   1:L PR[91] 10mm/sec CNT100;
   1:  PR[GP1:91,1] = PR[GP1:90,1] + 5.614;
   1:  PR[GP1:91,2] = PR[GP1:90,2] + -48.755;
   1:L PR[91] 10mm/sec CNT100;
   1:  PR[GP1:91,1] = PR[GP1:90,1] + 14.294;
   1:  PR[GP1:91,2] = PR[GP1:90,2] + -47.380;
   1:L PR[91] 10mm/sec CNT100;
   1:  PR[GP1:91,1] = PR[GP1:90,1] + 19.175;
   1:  PR[GP1:91,2] = PR[GP1:90,2] + -45.489;
   1:L PR[91] 10mm/sec CNT100;
   1:  PR[GP1:91,1] = PR[GP1:90,1] + 27.005;
   1:  PR[GP1:91,2] = PR[GP1:90,2] + -41.500;
   1:L PR[91] 10mm/sec CNT100;
   1:  PR[GP1:91,1] = PR[GP1:90,1] + 31.277;
   1:  PR[GP1:91,2] = PR[GP1:90,2] + -38.475;
   1:L PR[91] 10mm/sec CNT100;
   1:  PR[GP1:91,1] = PR[GP1:90,1] + 37.487;
   1:  PR[GP1:91,2] = PR[GP1:90,2] + -32.264;
   1:L PR[91] 10mm/sec CNT100;
   1:  PR[GP1:91,1] = PR[GP1:90,1] + 41.251;
   1:  PR[GP1:91,2] = PR[GP1:90,2] + -27.730;
   1:L PR[91] 10mm/sec CNT100;
   1:  PR[GP1:91,1] = PR[GP1:90,1] + 45.236;
   1:  PR[GP1:91,2] = PR[GP1:90,2] + -19.908;
   1:L PR[91] 10mm/sec CNT100;
   1:  PR[GP1:91,1] = PR[GP1:90,1] + 47.614;
   1:  PR[GP1:91,2] = PR[GP1:90,2] + -14.522;
   1:L PR[91] 10mm/sec CNT100;
   1:  PR[GP1:91,1] = PR[GP1:90,1] + 48.431;
   1:  PR[GP1:91,2] = PR[GP1:90,2] + -8.669;
   1:L PR[91] 10mm/sec CNT100;
   1:  PR[GP1:91,1] = PR[GP1:90,1] + 49.804;
   1:  PR[GP1:91,2] = PR[GP1:90,2] + 0.001;
   1:L PR[91] 10mm/sec CNT100;
   1:  PR[GP1:91,1] = PR[GP1:90,1] + 48.990;
   1:  PR[GP1:91,2] = PR[GP1:90,2] + 5.838;
   1:L PR[91] 10mm/sec CNT100;
   1:  PR[GP1:91,1] = PR[GP1:90,1] + 47.616;
   1:  PR[GP1:91,2] = PR[GP1:90,2] + 14.508;
   1:L PR[91] 10mm/sec CNT100;
   1:  PR[GP1:91,1] = PR[GP1:90,1] + 45.236;
   1:  PR[GP1:91,2] = PR[GP1:90,2] + 19.899;
   1:L PR[91] 10mm/sec CNT100;
   1:  PR[GP1:91,1] = PR[GP1:90,1] + 41.251;
   1:  PR[GP1:91,2] = PR[GP1:90,2] + 27.721;
   1:L PR[91] 10mm/sec CNT100;
   1:  PR[GP1:91,1] = PR[GP1:90,1] + 37.487;
   1:  PR[GP1:91,2] = PR[GP1:90,2] + 32.256;
   1:L PR[91] 10mm/sec CNT100;
   1:  PR[GP1:91,1] = PR[GP1:90,1] + 31.277;
   1:  PR[GP1:91,2] = PR[GP1:90,2] + 38.466;
   1:L PR[91] 10mm/sec CNT100;
   1:  PR[GP1:91,1] = PR[GP1:90,1] + 27.005;
   1:  PR[GP1:91,2] = PR[GP1:90,2] + 41.491;
   1:L PR[91] 10mm/sec CNT100;
   1:  PR[GP1:91,1] = PR[GP1:90,1] + 19.175;
   1:  PR[GP1:91,2] = PR[GP1:90,2] + 45.481;
   1:L PR[91] 10mm/sec CNT100;
   1:  PR[GP1:91,1] = PR[GP1:90,1] + 14.294;
   1:  PR[GP1:91,2] = PR[GP1:90,2] + 47.372;
   1:L PR[91] 10mm/sec CNT100;
   1:  PR[GP1:91,1] = PR[GP1:90,1] + 5.614;
   1:  PR[GP1:91,2] = PR[GP1:90,2] + 48.746;
   1:L PR[91] 10mm/sec CNT100;
   1:  PR[GP1:91,1] = PR[GP1:90,1] + 0.409;
   1:  PR[GP1:91,2] = PR[GP1:90,2] + 49.391;
   1:L PR[91] 10mm/sec CNT100;
   1:  PR[GP1:91,1] = PR[GP1:90,1] + -3.172;
   1:  PR[GP1:91,2] = PR[GP1:90,2] + 48.947;
   1:  PR[GP1:91,3] = PR[GP1:90,3] + 135.660;
   1:L PR[91] 10mm/sec CNT100;
   1:  PR[GP1:91,1] = PR[GP1:90,1] + -13.907;
   1:  PR[GP1:91,2] = PR[GP1:90,2] + 47.247;
   1:L PR[91] 10mm/sec CNT100;
   1:  PR[GP1:91,1] = PR[GP1:90,1] + -17.262;
   1:  PR[GP1:91,2] = PR[GP1:90,2] + 45.947;
   1:L PR[91] 10mm/sec CNT100;
   1:  PR[GP1:91,1] = PR[GP1:90,1] + -26.946;
   1:  PR[GP1:91,2] = PR[GP1:90,2] + 41.012;
   1:L PR[91] 10mm/sec CNT100;
   1:  PR[GP1:91,1] = PR[GP1:90,1] + -29.883;
   1:  PR[GP1:91,2] = PR[GP1:90,2] + 38.933;
   1:L PR[91] 10mm/sec CNT100;
   1:  PR[GP1:91,1] = PR[GP1:90,1] + -37.565;
   1:  PR[GP1:91,2] = PR[GP1:90,2] + 31.250;
   1:L PR[91] 10mm/sec CNT100;
   1:  PR[GP1:91,1] = PR[GP1:90,1] + -40.156;
   1:  PR[GP1:91,2] = PR[GP1:90,2] + 28.130;
   1:L PR[91] 10mm/sec CNT100;
   1:  PR[GP1:91,1] = PR[GP1:90,1] + -45.086;
   1:  PR[GP1:91,2] = PR[GP1:90,2] + 18.454;
   1:L PR[91] 10mm/sec CNT100;
   1:  PR[GP1:91,1] = PR[GP1:90,1] + -46.722;
   1:  PR[GP1:91,2] = PR[GP1:90,2] + 14.749;
   1:L PR[91] 10mm/sec CNT100;
   1:  PR[GP1:91,1] = PR[GP1:90,1] + -47.284;
   1:  PR[GP1:91,2] = PR[GP1:90,2] + 10.715;
   1:L PR[91] 10mm/sec CNT100;
   1:  PR[GP1:91,1] = PR[GP1:90,1] + -48.983;
   1:  PR[GP1:91,2] = PR[GP1:90,2] + -0.010;
   1:L PR[91] 10mm/sec CNT100;
   1:  PR[GP1:91,1] = PR[GP1:90,1] + -48.423;
   1:  PR[GP1:91,2] = PR[GP1:90,2] + -4.028;
   1:L PR[91] 10mm/sec CNT100;
   1:  PR[GP1:91,1] = PR[GP1:90,1] + -46.724;
   1:  PR[GP1:91,2] = PR[GP1:90,2] + -14.753;
   1:L PR[91] 10mm/sec CNT100;
   1:  PR[GP1:91,1] = PR[GP1:90,1] + -45.086;
   1:  PR[GP1:91,2] = PR[GP1:90,2] + -18.463;
   1:L PR[91] 10mm/sec CNT100;
   1:  PR[GP1:91,1] = PR[GP1:90,1] + -40.156;
   1:  PR[GP1:91,2] = PR[GP1:90,2] + -28.139;
   1:L PR[91] 10mm/sec CNT100;
   1:  PR[GP1:91,1] = PR[GP1:90,1] + -37.565;
   1:  PR[GP1:91,2] = PR[GP1:90,2] + -31.259;
   1:L PR[91] 10mm/sec CNT100;
   1:  PR[GP1:91,1] = PR[GP1:90,1] + -29.883;
   1:  PR[GP1:91,2] = PR[GP1:90,2] + -38.942;
   1:L PR[91] 10mm/sec CNT100;
   1:  PR[GP1:91,1] = PR[GP1:90,1] + -26.946;
   1:  PR[GP1:91,2] = PR[GP1:90,2] + -41.021;
   1:L PR[91] 10mm/sec CNT100;
   1:  PR[GP1:91,1] = PR[GP1:90,1] + -17.262;
   1:  PR[GP1:91,2] = PR[GP1:90,2] + -45.955;
   1:L PR[91] 10mm/sec CNT100;
   1:  PR[GP1:91,1] = PR[GP1:90,1] + -13.916;
   1:  PR[GP1:91,2] = PR[GP1:90,2] + -47.252;
   1:L PR[91] 10mm/sec CNT100;
   1:  PR[GP1:91,1] = PR[GP1:90,1] + -10.314;
   1:  PR[GP1:91,2] = PR[GP1:90,2] + -47.698;
   1:L PR[91] 10mm/sec CNT100;
   1:  PR[GP1:91,1] = PR[GP1:90,1] + 0.420;
   1:  PR[GP1:91,2] = PR[GP1:90,2] + -49.399;
   1:L PR[91] 10mm/sec CNT100;
   1:  PR[GP1:91,1] = PR[GP1:90,1] + 3.992;
   1:  PR[GP1:91,2] = PR[GP1:90,2] + -48.956;
   1:L PR[91] 10mm/sec CNT100;
   1:  PR[GP1:91,1] = PR[GP1:90,1] + 14.727;
   1:  PR[GP1:91,2] = PR[GP1:90,2] + -47.256;
   1:L PR[91] 10mm/sec CNT100;
   1:  PR[GP1:91,1] = PR[GP1:90,1] + 18.083;
   1:  PR[GP1:91,2] = PR[GP1:90,2] + -45.956;
   1:L PR[91] 10mm/sec CNT100;
   1:  PR[GP1:91,1] = PR[GP1:90,1] + 27.767;
   1:  PR[GP1:91,2] = PR[GP1:90,2] + -41.021;
   1:L PR[91] 10mm/sec CNT100;
   1:  PR[GP1:91,1] = PR[GP1:90,1] + 30.704;
   1:  PR[GP1:91,2] = PR[GP1:90,2] + -38.941;
   1:L PR[91] 10mm/sec CNT100;
   1:  PR[GP1:91,1] = PR[GP1:90,1] + 38.386;
   1:  PR[GP1:91,2] = PR[GP1:90,2] + -31.259;
   1:L PR[91] 10mm/sec CNT100;
   1:  PR[GP1:91,1] = PR[GP1:90,1] + 40.977;
   1:  PR[GP1:91,2] = PR[GP1:90,2] + -28.139;
   1:L PR[91] 10mm/sec CNT100;
   1:  PR[GP1:91,1] = PR[GP1:90,1] + 45.907;
   1:  PR[GP1:91,2] = PR[GP1:90,2] + -18.463;
   1:L PR[91] 10mm/sec CNT100;
   1:  PR[GP1:91,1] = PR[GP1:90,1] + 47.542;
   1:  PR[GP1:91,2] = PR[GP1:90,2] + -14.758;
   1:L PR[91] 10mm/sec CNT100;
   1:  PR[GP1:91,1] = PR[GP1:90,1] + 48.105;
   1:  PR[GP1:91,2] = PR[GP1:90,2] + -10.724;
   1:L PR[91] 10mm/sec CNT100;
   1:  PR[GP1:91,1] = PR[GP1:90,1] + 49.804;
   1:  PR[GP1:91,2] = PR[GP1:90,2] + 0.001;
   1:L PR[91] 10mm/sec CNT100;
   1:  PR[GP1:91,1] = PR[GP1:90,1] + 49.243;
   1:  PR[GP1:91,2] = PR[GP1:90,2] + 4.019;
   1:L PR[91] 10mm/sec CNT100;
   1:  PR[GP1:91,1] = PR[GP1:90,1] + 47.545;
   1:  PR[GP1:91,2] = PR[GP1:90,2] + 14.744;
   1:L PR[91] 10mm/sec CNT100;
   1:  PR[GP1:91,1] = PR[GP1:90,1] + 45.907;
   1:  PR[GP1:91,2] = PR[GP1:90,2] + 18.454;
   1:L PR[91] 10mm/sec CNT100;
   1:  PR[GP1:91,1] = PR[GP1:90,1] + 40.977;
   1:  PR[GP1:91,2] = PR[GP1:90,2] + 28.130;
   1:L PR[91] 10mm/sec CNT100;
   1:  PR[GP1:91,1] = PR[GP1:90,1] + 38.386;
   1:  PR[GP1:91,2] = PR[GP1:90,2] + 31.251;
   1:L PR[91] 10mm/sec CNT100;
   1:  PR[GP1:91,1] = PR[GP1:90,1] + 30.704;
   1:  PR[GP1:91,2] = PR[GP1:90,2] + 38.932;
   1:L PR[91] 10mm/sec CNT100;
   1:  PR[GP1:91,1] = PR[GP1:90,1] + 27.767;
   1:  PR[GP1:91,2] = PR[GP1:90,2] + 41.012;
   1:L PR[91] 10mm/sec CNT100;
   1:  PR[GP1:91,1] = PR[GP1:90,1] + 18.083;
   1:  PR[GP1:91,2] = PR[GP1:90,2] + 45.947;
   1:L PR[91] 10mm/sec CNT100;
   1:  PR[GP1:91,1] = PR[GP1:90,1] + 14.727;
   1:  PR[GP1:91,2] = PR[GP1:90,2] + 47.247;
   1:L PR[91] 10mm/sec CNT100;
   1:  PR[GP1:91,1] = PR[GP1:90,1] + 3.992;
   1:  PR[GP1:91,2] = PR[GP1:90,2] + 48.947;
   1:L PR[91] 10mm/sec CNT100;
   1:  PR[GP1:91,1] = PR[GP1:90,1] + 0.410;
   1:  PR[GP1:91,2] = PR[GP1:90,2] + 49.391;
   1:L PR[91] 10mm/sec CNT100;
   1:  PR[GP1:91,1] = PR[GP1:90,1] + -1.550;
   1:  PR[GP1:91,2] = PR[GP1:90,2] + 49.148;
   1:  PR[GP1:91,3] = PR[GP1:90,3] + 136.990;
   1:L PR[91] 10mm/sec CNT100;
   1:  PR[GP1:91,1] = PR[GP1:90,1] + -14.339;
   1:  PR[GP1:91,2] = PR[GP1:90,2] + 47.123;
   1:L PR[91] 10mm/sec CNT100;
   1:  PR[GP1:91,1] = PR[GP1:90,1] + -16.170;
   1:  PR[GP1:91,2] = PR[GP1:90,2] + 46.413;
   1:L PR[91] 10mm/sec CNT100;
   1:  PR[GP1:91,1] = PR[GP1:90,1] + -27.708;
   1:  PR[GP1:91,2] = PR[GP1:90,2] + 40.534;
   1:L PR[91] 10mm/sec CNT100;
   1:  PR[GP1:91,1] = PR[GP1:90,1] + -29.311;
   1:  PR[GP1:91,2] = PR[GP1:90,2] + 39.399;
   1:L PR[91] 10mm/sec CNT100;
   1:  PR[GP1:91,1] = PR[GP1:90,1] + -38.464;
   1:  PR[GP1:91,2] = PR[GP1:90,2] + 30.246;
   1:L PR[91] 10mm/sec CNT100;
   1:  PR[GP1:91,1] = PR[GP1:90,1] + -39.882;
   1:  PR[GP1:91,2] = PR[GP1:90,2] + 28.538;
   1:L PR[91] 10mm/sec CNT100;
   1:  PR[GP1:91,1] = PR[GP1:90,1] + -45.756;
   1:  PR[GP1:91,2] = PR[GP1:90,2] + 17.009;
   1:L PR[91] 10mm/sec CNT100;
   1:  PR[GP1:91,1] = PR[GP1:90,1] + -46.650;
   1:  PR[GP1:91,2] = PR[GP1:90,2] + 14.984;
   1:L PR[91] 10mm/sec CNT100;
   1:  PR[GP1:91,1] = PR[GP1:90,1] + -46.959;
   1:  PR[GP1:91,2] = PR[GP1:90,2] + 12.770;
   1:L PR[91] 10mm/sec CNT100;
   1:  PR[GP1:91,1] = PR[GP1:90,1] + -48.983;
   1:  PR[GP1:91,2] = PR[GP1:90,2] + -0.010;
   1:L PR[91] 10mm/sec CNT100;
   1:  PR[GP1:91,1] = PR[GP1:90,1] + -48.676;
   1:  PR[GP1:91,2] = PR[GP1:90,2] + -2.208;
   1:L PR[91] 10mm/sec CNT100;
   1:  PR[GP1:91,1] = PR[GP1:90,1] + -46.652;
   1:  PR[GP1:91,2] = PR[GP1:90,2] + -14.988;
   1:L PR[91] 10mm/sec CNT100;
   1:  PR[GP1:91,1] = PR[GP1:90,1] + -45.756;
   1:  PR[GP1:91,2] = PR[GP1:90,2] + -17.018;
   1:L PR[91] 10mm/sec CNT100;
   1:  PR[GP1:91,1] = PR[GP1:90,1] + -39.882;
   1:  PR[GP1:91,2] = PR[GP1:90,2] + -28.547;
   1:L PR[91] 10mm/sec CNT100;
   1:  PR[GP1:91,1] = PR[GP1:90,1] + -38.464;
   1:  PR[GP1:91,2] = PR[GP1:90,2] + -30.255;
   1:L PR[91] 10mm/sec CNT100;
   1:  PR[GP1:91,1] = PR[GP1:90,1] + -29.311;
   1:  PR[GP1:91,2] = PR[GP1:90,2] + -39.408;
   1:L PR[91] 10mm/sec CNT100;
   1:  PR[GP1:91,1] = PR[GP1:90,1] + -27.708;
   1:  PR[GP1:91,2] = PR[GP1:90,2] + -40.543;
   1:L PR[91] 10mm/sec CNT100;
   1:  PR[GP1:91,1] = PR[GP1:90,1] + -16.170;
   1:  PR[GP1:91,2] = PR[GP1:90,2] + -46.422;
   1:L PR[91] 10mm/sec CNT100;
   1:  PR[GP1:91,1] = PR[GP1:90,1] + -14.349;
   1:  PR[GP1:91,2] = PR[GP1:90,2] + -47.128;
   1:L PR[91] 10mm/sec CNT100;
   1:  PR[GP1:91,1] = PR[GP1:90,1] + -12.369;
   1:  PR[GP1:91,2] = PR[GP1:90,2] + -47.373;
   1:L PR[91] 10mm/sec CNT100;
   1:  PR[GP1:91,1] = PR[GP1:90,1] + 0.420;
   1:  PR[GP1:91,2] = PR[GP1:90,2] + -49.399;
   1:L PR[91] 10mm/sec CNT100;
   1:  PR[GP1:91,1] = PR[GP1:90,1] + 2.370;
   1:  PR[GP1:91,2] = PR[GP1:90,2] + -49.157;
   1:L PR[91] 10mm/sec CNT100;
   1:  PR[GP1:91,1] = PR[GP1:90,1] + 15.159;
   1:  PR[GP1:91,2] = PR[GP1:90,2] + -47.131;
   1:L PR[91] 10mm/sec CNT100;
   1:  PR[GP1:91,1] = PR[GP1:90,1] + 16.991;
   1:  PR[GP1:91,2] = PR[GP1:90,2] + -46.422;
   1:L PR[91] 10mm/sec CNT100;
   1:  PR[GP1:91,1] = PR[GP1:90,1] + 28.529;
   1:  PR[GP1:91,2] = PR[GP1:90,2] + -40.543;
   1:L PR[91] 10mm/sec CNT100;
   1:  PR[GP1:91,1] = PR[GP1:90,1] + 30.132;
   1:  PR[GP1:91,2] = PR[GP1:90,2] + -39.408;
   1:L PR[91] 10mm/sec CNT100;
   1:  PR[GP1:91,1] = PR[GP1:90,1] + 39.285;
   1:  PR[GP1:91,2] = PR[GP1:90,2] + -30.255;
   1:L PR[91] 10mm/sec CNT100;
   1:  PR[GP1:91,1] = PR[GP1:90,1] + 40.702;
   1:  PR[GP1:91,2] = PR[GP1:90,2] + -28.547;
   1:L PR[91] 10mm/sec CNT100;
   1:  PR[GP1:91,1] = PR[GP1:90,1] + 46.577;
   1:  PR[GP1:91,2] = PR[GP1:90,2] + -17.018;
   1:L PR[91] 10mm/sec CNT100;
   1:  PR[GP1:91,1] = PR[GP1:90,1] + 47.471;
   1:  PR[GP1:91,2] = PR[GP1:90,2] + -14.993;
   1:L PR[91] 10mm/sec CNT100;
   1:  PR[GP1:91,1] = PR[GP1:90,1] + 47.780;
   1:  PR[GP1:91,2] = PR[GP1:90,2] + -12.779;
   1:L PR[91] 10mm/sec CNT100;
   1:  PR[GP1:91,1] = PR[GP1:90,1] + 49.804;
   1:  PR[GP1:91,2] = PR[GP1:90,2] + 0.001;
   1:L PR[91] 10mm/sec CNT100;
   1:  PR[GP1:91,1] = PR[GP1:90,1] + 49.497;
   1:  PR[GP1:91,2] = PR[GP1:90,2] + 2.199;
   1:L PR[91] 10mm/sec CNT100;
   1:  PR[GP1:91,1] = PR[GP1:90,1] + 47.473;
   1:  PR[GP1:91,2] = PR[GP1:90,2] + 14.979;
   1:L PR[91] 10mm/sec CNT100;
   1:  PR[GP1:91,1] = PR[GP1:90,1] + 46.577;
   1:  PR[GP1:91,2] = PR[GP1:90,2] + 17.009;
   1:L PR[91] 10mm/sec CNT100;
   1:  PR[GP1:91,1] = PR[GP1:90,1] + 40.702;
   1:  PR[GP1:91,2] = PR[GP1:90,2] + 28.538;
   1:L PR[91] 10mm/sec CNT100;
   1:  PR[GP1:91,1] = PR[GP1:90,1] + 39.285;
   1:  PR[GP1:91,2] = PR[GP1:90,2] + 30.246;
   1:L PR[91] 10mm/sec CNT100;
   1:  PR[GP1:91,1] = PR[GP1:90,1] + 30.132;
   1:  PR[GP1:91,2] = PR[GP1:90,2] + 39.399;
   1:L PR[91] 10mm/sec CNT100;
   1:  PR[GP1:91,1] = PR[GP1:90,1] + 28.529;
   1:  PR[GP1:91,2] = PR[GP1:90,2] + 40.534;
   1:L PR[91] 10mm/sec CNT100;
   1:  PR[GP1:91,1] = PR[GP1:90,1] + 16.991;
   1:  PR[GP1:91,2] = PR[GP1:90,2] + 46.413;
   1:L PR[91] 10mm/sec CNT100;
   1:  PR[GP1:91,1] = PR[GP1:90,1] + 15.159;
   1:  PR[GP1:91,2] = PR[GP1:90,2] + 47.123;
   1:L PR[91] 10mm/sec CNT100;
   1:  PR[GP1:91,1] = PR[GP1:90,1] + 2.370;
   1:  PR[GP1:91,2] = PR[GP1:90,2] + 49.148;
   1:L PR[91] 10mm/sec CNT100;
   1:  PR[GP1:91,1] = PR[GP1:90,1] + 0.410;
   1:  PR[GP1:91,2] = PR[GP1:90,2] + 49.391;
   1:L PR[91] 10mm/sec CNT100;
   1:  PR[GP1:91,1] = PR[GP1:90,1] + 0.073;
   1:  PR[GP1:91,2] = PR[GP1:90,2] + 49.349;
   1:  PR[GP1:91,3] = PR[GP1:90,3] + 138.320;
   1:L PR[91] 10mm/sec CNT100;
   1:  PR[GP1:91,1] = PR[GP1:90,1] + -14.771;
   1:  PR[GP1:91,2] = PR[GP1:90,2] + 46.998;
   1:L PR[91] 10mm/sec CNT100;
   1:  PR[GP1:91,1] = PR[GP1:90,1] + -15.079;
   1:  PR[GP1:91,2] = PR[GP1:90,2] + 46.879;
   1:L PR[91] 10mm/sec CNT100;
   1:  PR[GP1:91,1] = PR[GP1:90,1] + -28.470;
   1:  PR[GP1:91,2] = PR[GP1:90,2] + 40.056;
   1:L PR[91] 10mm/sec CNT100;
   1:  PR[GP1:91,1] = PR[GP1:90,1] + -28.739;
   1:  PR[GP1:91,2] = PR[GP1:90,2] + 39.865;
   1:L PR[91] 10mm/sec CNT100;
   1:  PR[GP1:91,1] = PR[GP1:90,1] + -39.363;
   1:  PR[GP1:91,2] = PR[GP1:90,2] + 29.241;
   1:L PR[91] 10mm/sec CNT100;
   1:  PR[GP1:91,1] = PR[GP1:90,1] + -39.607;
   1:  PR[GP1:91,2] = PR[GP1:90,2] + 28.947;
   1:L PR[91] 10mm/sec CNT100;
   1:  PR[GP1:91,1] = PR[GP1:90,1] + -46.426;
   1:  PR[GP1:91,2] = PR[GP1:90,2] + 15.564;
   1:L PR[91] 10mm/sec CNT100;
